KUKA KRL program: EPS_2_25694_GD02_A_20260114065900.src

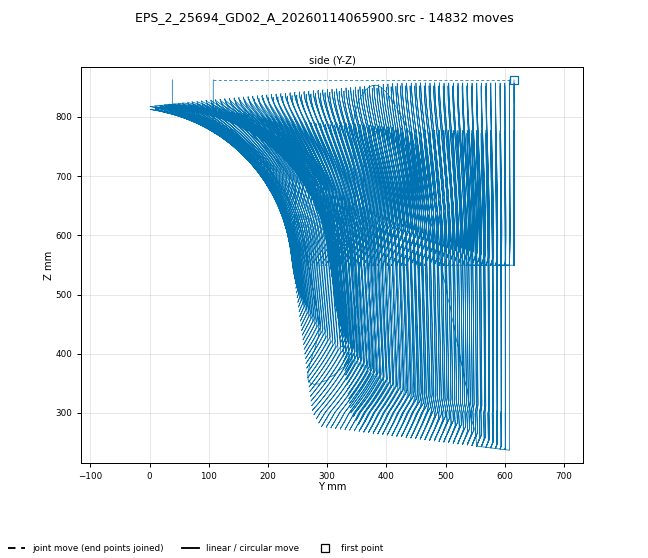
[picture p0: tool path of EPS_2_25694_GD02_A_20260114065900.src, 14832 of 14834 moves have a stored position in this frame; points joined in program order, loops and branches not executed]
&ACCESS RVP
&REL 4
&COMMENT QRS 19112012
&PARAM EDITMASK = *
DEF PART()
EXT BAS (BAS_COMMAND :IN,REAL :IN )
INT I
BAS (#INITMOV,0 )

;KUKA QRS Post kuka4.cps  Date:22-06-2017 !

File_ID=2962

QRS_PRE_INIT()

;Init var - Until changes are made in qrs_pre_init
Outlet_Square_prg=0
Inlet_1_Square_prg=0
Inlet_2_Square_prg=0
Inlet_3_Square_prg=0
Inlet_4_Square_prg=0
Inlet_5_Square_prg=0

Outlet_1={X 0.000, Y 425.000, Z 586.000, B 0.000, E1 0.000 }
Inlet_1={X 0.000, Y 466.000, Z 544.000, B 0.000, E1 154.000 }
Outlet_1_type=533
Inlet_1_type=457
;QRS#1=Sidecore dimensions
;QRS#2=525-21" Concrete
;QRS#3=450-18" Concrete
;QRS#4=
;QRS#5=
;QRS#6=
;QRS#7=
;QRS#8=
;QRS#9=S306-32
;QRS#10=28A PSX-2
;QRS#11=
;QRS#12=
;QRS#13=
;QRS#14=
;QRS#15=
;QRS#16=1220x127x1219 4'
;QRS#17=EPS Height
;QRS#18=852,5
;QRS#19=*
;QRS#20= UPDATED VERSION 22-06-2017
;QRS#21=*
Outlet_Square=0250
Inlet_1_Square=0250
Inlet_2_Square=0
Inlet_3_Square=0
Inlet_4_Square=0
Inlet_5_Square=0
Mill_Square=1
Outlet_Square_Prg=263
Inlet_1_Square_prg=274

QRS_INIT()

$ADVANCE=5

; T1
PTP {E1 172.625,E2 172.625}
PTP {X 0,Y 615.419,A -85,B 0,C 180,E1 172.625,E2 172.625,E3 0,E4 0,E5 0,E6 0}
QRS_SPEED_INIT()
LIN {X 0,Y 615.419,Z 862.5,A -85,B 0,C 180,E1 172.625,E2 172.625,E3 0,E4 0,E5 0,E6 0} C_VEL
LIN {X 0,Y 615.419,Z 551.53,A -85,B 0,C 180,E1 172.625,E2 172.625} C_VEL
LIN {X 0,Y 615.447,Z 549.53,A -85,B 0,C 180,E1 172.811,E2 172.811} C_VEL
LIN {X 0,Y 615.861,Z 549.53,A -85,B 0,C 180,E1 174.195,E2 174.195} C_VEL
LIN {X 0,Y 615.858,Z 549.53,A -85,B 0,C 180,E1 178.842,E2 178.842} C_VEL
LIN {X 0,Y 615.837,Z 549.53,A -85,B 0,C 180,E1 183.481,E2 183.481} C_VEL
LIN {X 0,Y 615.852,Z 549.53,A -85,B 0,C 180,E1 188.144,E2 188.144} C_VEL
LIN {X 0,Y 615.818,Z 549.53,A -85,B 0,C 180,E1 192.862,E2 192.862} C_VEL
LIN {X 0,Y 615.818,Z 549.53,A -85,B 0,C 180,E1 197.671,E2 197.671} C_VEL
LIN {X 0,Y 615.804,Z 549.53,A -85,B 0,C 180,E1 197.994,E2 197.994} C_VEL
LIN {X 0,Y 615.767,Z 549.53,A -85,B 0,C 180,E1 202.614,E2 202.614} C_VEL
LIN {X 0,Y 615.241,Z 549.53,A -85,B 0,C 180,E1 205.173,E2 205.173} C_VEL
LIN {X 0,Y 615.742,Z 549.53,A -85,B 0,C 180,E1 207.742,E2 207.742} C_VEL
LIN {X 0,Y 615.253,Z 549.53,A -85,B 0,C 180,E1 210.422,E2 210.422} C_VEL
LIN {X 0,Y 615.857,Z 549.53,A -85,B 0,C 180,E1 213.116,E2 213.116} C_VEL
LIN {X 0,Y 615.548,Z 549.53,A -85,B 0,C 180,E1 215.951,E2 215.951} C_VEL
LIN {X 0,Y 615.599,Z 549.53,A -85,B 0,C 180,E1 217.864,E2 217.864} C_VEL
LIN {X 0,Y 615.649,Z 549.53,A -85,B 0,C 180,E1 221.91,E2 221.91} C_VEL
LIN {X 0,Y 615.215,Z 549.53,A -85,B 0,C 180,E1 225.149,E2 225.149} C_VEL
LIN {X 0,Y 615.671,Z 549.53,A -85,B 0,C 180,E1 228.092,E2 228.092} C_VEL
LIN {X 0,Y 615.575,Z 549.53,A -85,B 0,C 180,E1 232.139,E2 232.139} C_VEL
LIN {X 0,Y 615.56,Z 549.53,A -85,B 0,C 180,E1 234.05,E2 234.05} C_VEL
LIN {X 0,Y 615.724,Z 549.53,A -85,B 0,C 180,E1 236.077,E2 236.077} C_VEL
LIN {X 0,Y 615.758,Z 549.53,A -85,B 0,C 180,E1 236.878,E2 236.878} C_VEL
LIN {X 0,Y 615.847,Z 549.53,A -85,B 0,C 180,E1 240.622,E2 240.622} C_VEL
LIN {X 0,Y 615.221,Z 549.53,A -85,B 0,C 180,E1 240.78,E2 240.78} C_VEL
LIN {X 0,Y 615.113,Z 550.032,A -85,B 0,C 180,E1 240.802,E2 240.802} C_VEL
LIN {X 0,Y 615.441,Z 600.013,A -85,B 0,C 180,E1 241.477,E2 241.477} C_VEL
LIN {X 0,Y 615.52,Z 611.103,A -85,B 0,C 180,E1 241.656,E2 241.656} C_VEL
LIN {X 0,Y 615.538,Z 625.601,A -85,B 0,C 180,E1 241.961,E2 241.961} C_VEL
LIN {X 0,Y 615.511,Z 635.884,A -85,B 0,C 180,E1 242.221,E2 242.221} C_VEL
LIN {X 0,Y 615.677,Z 651.48,A -85,B 0,C 180,E1 242.705,E2 242.705} C_VEL
LIN {X 0,Y 615.654,Z 663.918,A -85,B 0,C 180,E1 243.151,E2 243.151} C_VEL
LIN {X 0,Y 615.577,Z 673.836,A -85,B 0,C 180,E1 243.553,E2 243.553} C_VEL
LIN {X 0,Y 615.711,Z 689.57,A -85,B 0,C 180,E1 244.286,E2 244.286} C_VEL
LIN {X 0,Y 615.693,Z 701.923,A -85,B 0,C 180,E1 244.935,E2 244.935} C_VEL
LIN {X 0,Y 615.683,Z 713.602,A -85,B 0,C 180,E1 245.616,E2 245.616} C_VEL
LIN {X 0,Y 615.707,Z 725.064,A -85,B 0,C 180,E1 246.355,E2 246.355} C_VEL
LIN {X 0,Y 615.721,Z 736.37,A -85,B 0,C 180,E1 247.156,E2 247.156} C_VEL
LIN {X 0,Y 615.717,Z 747.376,A -85,B 0,C 180,E1 248.011,E2 248.011} C_VEL
LIN {X 0,Y 615.704,Z 756.639,A -85,B 0,C 180,E1 248.79,E2 248.79} C_VEL
LIN {X 0,Y 615.752,Z 766.777,A -85,B 0,C 180,E1 249.722,E2 249.722} C_VEL
LIN {X 0,Y 615.723,Z 776.042,A -85,B 0,C 180,E1 250.645,E2 250.645} C_VEL
LIN {X 0,Y 615.683,Z 784.412,A -85,B 0,C 180,E1 251.548,E2 251.548} C_VEL
LIN {X 0,Y 615.767,Z 792.766,A -85,B 0,C 180,E1 252.531,E2 252.531} C_VEL
LIN {X 0,Y 615.719,Z 800.672,A -85,B 0,C 180,E1 253.541,E2 253.541} C_VEL
LIN {X 0,Y 615.582,Z 807.418,A -85,B 0,C 180,E1 254.471,E2 254.471} C_VEL
LIN {X 0,Y 615.671,Z 815.053,A -85,B 0,C 180,E1 255.643,E2 255.643} C_VEL
LIN {X 0,Y 615.808,Z 820.43,A -85,B 0,C 180,E1 256.542,E2 256.542} C_VEL
LIN {X 0,Y 615.575,Z 826.903,A -85,B 0,C 180,E1 257.727,E2 257.727} C_VEL
LIN {X 0,Y 615.615,Z 832.619,A -85,B 0,C 180,E1 258.912,E2 258.912} C_VEL
LIN {X 0,Y 615.829,Z 837.629,A -85,B 0,C 180,E1 260.095,E2 260.095} C_VEL
LIN {X 0,Y 615.604,Z 842.059,A -85,B 0,C 180,E1 261.267,E2 261.267} C_VEL
LIN {X 0,Y 615.655,Z 846.467,A -85,B 0,C 180,E1 262.659,E2 262.659} C_VEL
LIN {X 0,Y 615.789,Z 849.367,A -85,B 0,C 180,E1 263.748,E2 263.748} C_VEL
LIN {X 0,Y 615.594,Z 851.398,A -85,B 0,C 180,E1 264.656,E2 264.656} C_VEL
LIN {X 0,Y 615.536,Z 853.159,A -85,B 0,C 180,E1 265.587,E2 265.587} C_VEL
LIN {X 0,Y 615.642,Z 854.59,A -85,B 0,C 180,E1 266.518,E2 266.518} C_VEL
LIN {X 0,Y 615.713,Z 856.053,A -85,B 0,C 180,E1 267.911,E2 267.911} C_VEL
LIN {X 0,Y 615.553,Z 856.714,A -85,B 0,C 180,E1 268.839,E2 268.839} C_VEL
LIN {X 0,Y 615.842,Z 856.659,A -85,B 0,C 180,E1 271.158,E2 271.158} C_VEL
LIN {X 0,Y 615.567,Z 855.719,A -85,B 0,C 180,E1 272.551,E2 272.551} C_VEL
LIN {X 0,Y 615.55,Z 854.61,A -85,B 0,C 180,E1 273.481,E2 273.481} C_VEL
LIN {X 0,Y 615.713,Z 853.131,A -85,B 0,C 180,E1 274.41,E2 274.41} C_VEL
LIN {X 0,Y 615.771,Z 851.372,A -85,B 0,C 180,E1 275.34,E2 275.34} C_VEL
LIN {X 0,Y 615.615,Z 849.407,A -85,B 0,C 180,E1 276.25,E2 276.25} C_VEL
LIN {X 0,Y 615.622,Z 846.269,A -85,B 0,C 180,E1 277.417,E2 277.417} C_VEL
LIN {X 0,Y 615.784,Z 842.039,A -85,B 0,C 180,E1 278.729,E2 278.729} C_VEL
LIN {X 0,Y 615.572,Z 837.675,A -85,B 0,C 180,E1 279.907,E2 279.907} C_VEL
LIN {X 0,Y 615.632,Z 832.626,A -85,B 0,C 180,E1 281.085,E2 281.085} C_VEL
LIN {X 0,Y 615.805,Z 826.888,A -85,B 0,C 180,E1 282.266,E2 282.266} C_VEL
LIN {X 0,Y 615.626,Z 820.461,A -85,B 0,C 180,E1 283.459,E2 283.459} C_VEL
LIN {X 0,Y 615.698,Z 813.201,A -85,B 0,C 180,E1 284.653,E2 284.653} C_VEL
LIN {X 0,Y 615.811,Z 807.636,A -85,B 0,C 180,E1 285.488,E2 285.488} C_VEL
LIN {X 0,Y 615.663,Z 798.205,A -85,B 0,C 180,E1 286.79,E2 286.79} C_VEL
LIN {X 0,Y 615.737,Z 789.613,A -85,B 0,C 180,E1 287.852,E2 287.852} C_VEL
LIN {X 0,Y 615.77,Z 781.421,A -85,B 0,C 180,E1 288.783,E2 288.783} C_VEL
LIN {X 0,Y 615.696,Z 771.534,A -85,B 0,C 180,E1 289.815,E2 289.815} C_VEL
LIN {X 0,Y 615.715,Z 763.548,A -85,B 0,C 180,E1 290.587,E2 290.587} C_VEL
LIN {X 0,Y 615.746,Z 753.046,A -85,B 0,C 180,E1 291.517,E2 291.517} C_VEL
LIN {X 0,Y 615.704,Z 743.056,A -85,B 0,C 180,E1 292.335,E2 292.335} C_VEL
LIN {X 0,Y 615.702,Z 733.306,A -85,B 0,C 180,E1 293.07,E2 293.07} C_VEL
LIN {X 0,Y 615.683,Z 721.643,A -85,B 0,C 180,E1 293.873,E2 293.873} C_VEL
LIN {X 0,Y 615.698,Z 709.605,A -85,B 0,C 180,E1 294.622,E2 294.622} C_VEL
LIN {X 0,Y 615.65,Z 698.907,A -85,B 0,C 180,E1 295.233,E2 295.233} C_VEL
LIN {X 0,Y 615.644,Z 688.043,A -85,B 0,C 180,E1 295.795,E2 295.795} C_VEL
LIN {X 0,Y 615.702,Z 673.896,A -85,B 0,C 180,E1 296.439,E2 296.439} C_VEL
LIN {X 0,Y 615.617,Z 660.697,A -85,B 0,C 180,E1 296.97,E2 296.97} C_VEL
LIN {X 0,Y 615.556,Z 651.549,A -85,B 0,C 180,E1 297.299,E2 297.299} C_VEL
LIN {X 0,Y 615.623,Z 634.845,A -85,B 0,C 180,E1 297.8,E2 297.8} C_VEL
LIN {X 0,Y 615.442,Z 622.425,A -85,B 0,C 180,E1 298.118,E2 298.118} C_VEL
LIN {X 0,Y 615.615,Z 610.181,A -85,B 0,C 180,E1 298.357,E2 298.357} C_VEL
LIN {X 0,Y 615.523,Z 589,A -85,B 0,C 180,E1 298.668,E2 298.668} C_VEL
LIN {X 0,Y 615.166,Z 549.53,A -85,B 0,C 180,E1 299.213,E2 299.213} C_VEL
LIN {X 0,Y 615.783,Z 549.53,A -85,B 0,C 180,E1 299.346,E2 299.346} C_VEL
LIN {X 0,Y 615.859,Z 549.53,A -85,B 0,C 180,E1 300.386,E2 300.386} C_VEL
LIN {X 0,Y 615.153,Z 549.53,A -85,B 0,C 180,E1 303.844,E2 303.844} C_VEL
LIN {X 0,Y 615.7,Z 549.53,A -85,B 0,C 180,E1 305.938,E2 305.938} C_VEL
LIN {X 0,Y 615.751,Z 549.53,A -85,B 0,C 180,E1 308.854,E2 308.854} C_VEL
LIN {X 0,Y 615.252,Z 549.53,A -85,B 0,C 180,E1 311.94,E2 311.94} C_VEL
LIN {X 0,Y 615.68,Z 549.53,A -85,B 0,C 180,E1 314.894,E2 314.894} C_VEL
LIN {X 0,Y 615.644,Z 549.53,A -85,B 0,C 180,E1 318.494,E2 318.494} C_VEL
LIN {X 0,Y 615.361,Z 549.53,A -85,B 0,C 180,E1 321.114,E2 321.114} C_VEL
LIN {X 0,Y 615.413,Z 549.53,A -85,B 0,C 180,E1 322.155,E2 322.155} C_VEL
LIN {X 0,Y 615.665,Z 549.53,A -85,B 0,C 180,E1 324.057,E2 324.057} C_VEL
LIN {X 0,Y 615.125,Z 549.53,A -85,B 0,C 180,E1 326.84,E2 326.84} C_VEL
LIN {X 0,Y 615.717,Z 549.53,A -85,B 0,C 180,E1 329.603,E2 329.603} C_VEL
LIN {X 0,Y 615.208,Z 549.53,A -85,B 0,C 180,E1 332.232,E2 332.232} C_VEL
LIN {X 0,Y 615.747,Z 549.53,A -85,B 0,C 180,E1 334.849,E2 334.849} C_VEL
LIN {X 0,Y 615.78,Z 549.53,A -85,B 0,C 180,E1 339.877,E2 339.877} C_VEL
LIN {X 0,Y 615.794,Z 549.53,A -85,B 0,C 180,E1 343.783,E2 343.783} C_VEL
LIN {X 0,Y 615.811,Z 549.53,A -85,B 0,C 180,E1 349.506,E2 349.506} C_VEL
LIN {X 0,Y 615.84,Z 549.53,A -85,B 0,C 180,E1 354.192,E2 354.192} C_VEL
LIN {X 0,Y 615.881,Z 549.53,A -85,B 0,C 180,E1 358.839,E2 358.839} C_VEL
LIN {X 0,Y 615.868,Z 549.53,A -85,B 0,C 180,E1 363.479,E2 363.479} C_VEL
LIN {X 0,Y 615.819,Z 549.53,A -85,B 0,C 180,E1 368.142,E2 368.142} C_VEL
LIN {X 0,Y 615.829,Z 549.53,A -85,B 0,C 180,E1 372.86,E2 372.86} C_VEL
LIN {X 0,Y 615.811,Z 549.53,A -85,B 0,C 180,E1 377.669,E2 377.669} C_VEL
LIN {X 0,Y 615.807,Z 549.53,A -85,B 0,C 180,E1 378.001,E2 378.001} C_VEL
LIN {X 0,Y 615.775,Z 549.53,A -85,B 0,C 180,E1 382.611,E2 382.611} C_VEL
LIN {X 0,Y 615.234,Z 549.53,A -85,B 0,C 180,E1 385.171,E2 385.171} C_VEL
LIN {X 0,Y 615.726,Z 549.53,A -85,B 0,C 180,E1 387.74,E2 387.74} C_VEL
LIN {X 0,Y 615.245,Z 549.53,A -85,B 0,C 180,E1 390.42,E2 390.42} C_VEL
LIN {X 0,Y 615.861,Z 549.53,A -85,B 0,C 180,E1 393.113,E2 393.113} C_VEL
LIN {X 0,Y 615.544,Z 549.53,A -85,B 0,C 180,E1 395.949,E2 395.949} C_VEL
LIN {X 0,Y 615.616,Z 549.53,A -85,B 0,C 180,E1 397.87,E2 397.87} C_VEL
LIN {X 0,Y 615.686,Z 549.53,A -85,B 0,C 180,E1 401.904,E2 401.904} C_VEL
LIN {X 0,Y 615.226,Z 549.53,A -85,B 0,C 180,E1 405.145,E2 405.145} C_VEL
LIN {X 0,Y 615.687,Z 549.53,A -85,B 0,C 180,E1 408.096,E2 408.096} C_VEL
LIN {X 0,Y 615.59,Z 549.53,A -85,B 0,C 180,E1 412.133,E2 412.133} C_VEL
LIN {X 0,Y 615.555,Z 549.53,A -85,B 0,C 180,E1 414.052,E2 414.052} C_VEL
LIN {X 0,Y 615.724,Z 549.53,A -85,B 0,C 180,E1 416.073,E2 416.073} C_VEL
LIN {X 0,Y 615.732,Z 549.53,A -85,B 0,C 180,E1 416.879,E2 416.879} C_VEL
LIN {X 0,Y 615.544,Z 549.53,A -85,B 0,C 180,E1 420.514,E2 420.514} C_VEL
LIN {X 0,Y 615.505,Z 549.53,A -85,B 0,C 180,E1 422.249,E2 422.249} C_VEL
LIN {X 0,Y 615.421,Z 549.53,A -85,B 0,C 180,E1 425.664,E2 425.664} C_VEL
LIN {X 0,Y 615.586,Z 549.53,A -85,B 0,C 180,E1 427.382,E2 427.382} C_VEL
LIN {X 0,Y 615.803,Z 549.53,A -85,B 0,C 180,E1 431.999,E2 431.999} C_VEL
LIN {X 0,Y 615.813,Z 549.53,A -85,B 0,C 180,E1 432.331,E2 432.331} C_VEL
LIN {X 0,Y 615.817,Z 549.53,A -85,B 0,C 180,E1 437.14,E2 437.14} C_VEL
LIN {X 0,Y 615.839,Z 549.53,A -85,B 0,C 180,E1 441.858,E2 441.858} C_VEL
LIN {X 0,Y 615.871,Z 549.53,A -85,B 0,C 180,E1 446.521,E2 446.521} C_VEL
LIN {X 0,Y 615.493,Z 549.53,A -85,B 0,C 180,E1 448.841,E2 448.841} C_VEL
LIN {X 0,Y 615.592,Z 549.53,A -85,B 0,C 180,E1 451.161,E2 451.161} C_VEL
LIN {X 0,Y 615.322,Z 549.53,A -85,B 0,C 180,E1 451.292,E2 451.292} C_VEL
LIN {X 0,Y 615.521,Z 551.584,A -85,B 0,C 180,E1 451.335,E2 451.335} C_VEL
LIN {X 0,Y 615.568,Z 564.334,A -85,B 0,C 180,E1 451.538,E2 451.538} C_VEL
LIN {X 0,Y 615.674,Z 576.042,A -85,B 0,C 180,E1 451.784,E2 451.784} C_VEL
LIN {X 0,Y 615.724,Z 587.841,A -85,B 0,C 180,E1 452.089,E2 452.089} C_VEL
LIN {X 0,Y 615.604,Z 599.369,A -85,B 0,C 180,E1 452.437,E2 452.437} C_VEL
LIN {X 0,Y 615.735,Z 610.571,A -85,B 0,C 180,E1 452.843,E2 452.843} C_VEL
LIN {X 0,Y 615.763,Z 621.858,A -85,B 0,C 180,E1 453.307,E2 453.307} C_VEL
LIN {X 0,Y 615.701,Z 631.978,A -85,B 0,C 180,E1 453.773,E2 453.773} C_VEL
LIN {X 0,Y 615.733,Z 642.117,A -85,B 0,C 180,E1 454.295,E2 454.295} C_VEL
LIN {X 0,Y 615.752,Z 652.294,A -85,B 0,C 180,E1 454.877,E2 454.877} C_VEL
LIN {X 0,Y 615.751,Z 663.293,A -85,B 0,C 180,E1 455.576,E2 455.576} C_VEL
LIN {X 0,Y 615.738,Z 671.827,A -85,B 0,C 180,E1 456.167,E2 456.167} C_VEL
LIN {X 0,Y 615.744,Z 681.127,A -85,B 0,C 180,E1 456.874,E2 456.874} C_VEL
LIN {X 0,Y 615.757,Z 689.335,A -85,B 0,C 180,E1 457.55,E2 457.55} C_VEL
LIN {X 0,Y 615.801,Z 697.599,A -85,B 0,C 180,E1 458.291,E2 458.291} C_VEL
LIN {X 0,Y 615.737,Z 706.589,A -85,B 0,C 180,E1 459.172,E2 459.172} C_VEL
LIN {X 0,Y 615.734,Z 713.495,A -85,B 0,C 180,E1 459.907,E2 459.907} C_VEL
LIN {X 0,Y 615.829,Z 721.068,A -85,B 0,C 180,E1 460.789,E2 460.789} C_VEL
LIN {X 0,Y 615.72,Z 728.094,A -85,B 0,C 180,E1 461.677,E2 461.677} C_VEL
LIN {X 0,Y 615.671,Z 734.517,A -85,B 0,C 180,E1 462.568,E2 462.568} C_VEL
LIN {X 0,Y 615.768,Z 740.348,A -85,B 0,C 180,E1 463.459,E2 463.459} C_VEL
LIN {X 0,Y 615.748,Z 745.727,A -85,B 0,C 180,E1 464.355,E2 464.355} C_VEL
LIN {X 0,Y 615.626,Z 750.659,A -85,B 0,C 180,E1 465.258,E2 465.258} C_VEL
LIN {X 0,Y 615.725,Z 756.396,A -85,B 0,C 180,E1 466.459,E2 466.459} C_VEL
LIN {X 0,Y 615.801,Z 759.837,A -85,B 0,C 180,E1 467.266,E2 467.266} C_VEL
LIN {X 0,Y 615.629,Z 764.32,A -85,B 0,C 180,E1 468.452,E2 468.452} C_VEL
LIN {X 0,Y 615.688,Z 767.676,A -85,B 0,C 180,E1 469.51,E2 469.51} C_VEL
LIN {X 0,Y 615.806,Z 769.293,A -85,B 0,C 180,E1 470.122,E2 470.122} C_VEL
LIN {X 0,Y 615.749,Z 770.875,A -85,B 0,C 180,E1 470.743,E2 470.743} C_VEL
LIN {X 0,Y 615.585,Z 773.45,A -85,B 0,C 180,E1 471.994,E2 471.994} C_VEL
LIN {X 0,Y 615.622,Z 774.496,A -85,B 0,C 180,E1 472.619,E2 472.619} C_VEL
LIN {X 0,Y 615.769,Z 775.581,A -85,B 0,C 180,E1 473.516,E2 473.516} C_VEL
LIN {X 0,Y 615.695,Z 776.356,A -85,B 0,C 180,E1 474.392,E2 474.392} C_VEL
LIN {X 0,Y 615.585,Z 776.792,A -85,B 0,C 180,E1 475.158,E2 475.158} C_VEL
LIN {X 0,Y 615.649,Z 776.852,A -85,B 0,C 180,E1 476.443,E2 476.443} C_VEL
LIN {X 0,Y 615.764,Z 776.185,A -85,B 0,C 180,E1 477.74,E2 477.74} C_VEL
LIN {X 0,Y 615.646,Z 775.322,A -85,B 0,C 180,E1 478.631,E2 478.631} C_VEL
LIN {X 0,Y 615.648,Z 774.08,A -85,B 0,C 180,E1 479.534,E2 479.534} C_VEL
LIN {X 0,Y 615.799,Z 772.553,A -85,B 0,C 180,E1 480.392,E2 480.392} C_VEL
LIN {X 0,Y 615.717,Z 770.538,A -85,B 0,C 180,E1 481.325,E2 481.325} C_VEL
LIN {X 0,Y 615.599,Z 768.043,A -85,B 0,C 180,E1 482.27,E2 482.27} C_VEL
LIN {X 0,Y 615.707,Z 763.994,A -85,B 0,C 180,E1 483.548,E2 483.548} C_VEL
LIN {X 0,Y 615.783,Z 760.587,A -85,B 0,C 180,E1 484.456,E2 484.456} C_VEL
LIN {X 0,Y 615.616,Z 755.31,A -85,B 0,C 180,E1 485.698,E2 485.698} C_VEL
LIN {X 0,Y 615.727,Z 749.175,A -85,B 0,C 180,E1 486.921,E2 486.921} C_VEL
LIN {X 0,Y 615.826,Z 745.732,A -85,B 0,C 180,E1 487.551,E2 487.551} C_VEL
LIN {X 0,Y 615.668,Z 739.293,A -85,B 0,C 180,E1 488.626,E2 488.626} C_VEL
LIN {X 0,Y 615.685,Z 733.233,A -85,B 0,C 180,E1 489.533,E2 489.533} C_VEL
LIN {X 0,Y 615.809,Z 725.413,A -85,B 0,C 180,E1 490.581,E2 490.581} C_VEL
LIN {X 0,Y 615.706,Z 717.809,A -85,B 0,C 180,E1 491.512,E2 491.512} C_VEL
LIN {X 0,Y 615.692,Z 710.996,A -85,B 0,C 180,E1 492.278,E2 492.278} C_VEL
LIN {X 0,Y 615.759,Z 703.806,A -85,B 0,C 180,E1 493.022,E2 493.022} C_VEL
LIN {X 0,Y 615.754,Z 694.645,A -85,B 0,C 180,E1 493.889,E2 493.889} C_VEL
LIN {X 0,Y 615.725,Z 686.193,A -85,B 0,C 180,E1 494.624,E2 494.624} C_VEL
LIN {X 0,Y 615.738,Z 677.048,A -85,B 0,C 180,E1 495.352,E2 495.352} C_VEL
LIN {X 0,Y 615.745,Z 668.071,A -85,B 0,C 180,E1 496.009,E2 496.009} C_VEL
LIN {X 0,Y 615.751,Z 658.065,A -85,B 0,C 180,E1 496.675,E2 496.675} C_VEL
LIN {X 0,Y 615.747,Z 648.614,A -85,B 0,C 180,E1 497.249,E2 497.249} C_VEL
LIN {X 0,Y 615.67,Z 638.444,A -85,B 0,C 180,E1 497.812,E2 497.812} C_VEL
LIN {X 0,Y 615.756,Z 627.627,A -85,B 0,C 180,E1 498.343,E2 498.343} C_VEL
LIN {X 0,Y 615.751,Z 616.912,A -85,B 0,C 180,E1 498.815,E2 498.815} C_VEL
LIN {X 0,Y 615.675,Z 606.253,A -85,B 0,C 180,E1 499.232,E2 499.232} C_VEL
LIN {X 0,Y 615.684,Z 596.594,A -85,B 0,C 180,E1 499.564,E2 499.564} C_VEL
LIN {X 0,Y 615.68,Z 583.685,A -85,B 0,C 180,E1 499.938,E2 499.938} C_VEL
LIN {X 0,Y 615.56,Z 573.065,A -85,B 0,C 180,E1 500.2,E2 500.2} C_VEL
LIN {X 0,Y 615.621,Z 560.618,A -85,B 0,C 180,E1 500.436,E2 500.436} C_VEL
LIN {X 0,Y 615.473,Z 550.692,A -85,B 0,C 180,E1 500.59,E2 500.59} C_VEL
LIN {X 0,Y 615.123,Z 549.53,A -85,B 0,C 180,E1 500.623,E2 500.623} C_VEL
LIN {X 0,Y 615.755,Z 549.53,A -85,B 0,C 180,E1 500.83,E2 500.83} C_VEL
LIN {X 0,Y 615.851,Z 549.53,A -85,B 0,C 180,E1 501.154,E2 501.154} C_VEL
LIN {X 0,Y 615.701,Z 549.53,A -85,B 0,C 180,E1 504.062,E2 504.062} C_VEL
LIN {X 0,Y 615.123,Z 549.53,A -85,B 0,C 180,E1 506.842,E2 506.842} C_VEL
LIN {X 0,Y 615.677,Z 549.53,A -85,B 0,C 180,E1 509.604,E2 509.604} C_VEL
LIN {X 0,Y 615.181,Z 549.53,A -85,B 0,C 180,E1 512.234,E2 512.234} C_VEL
LIN {X 0,Y 615.722,Z 549.53,A -85,B 0,C 180,E1 514.85,E2 514.85} C_VEL
LIN {X 0,Y 615.796,Z 549.53,A -85,B 0,C 180,E1 519.88,E2 519.88} C_VEL
LIN {X 0,Y 615.742,Z 549.53,A -85,B 0,C 180,E1 523.3,E2 523.3} C_VEL
LIN {X 0,Y 615.403,Z 549.53,A -85,B 0,C 180,E1 524.739,E2 524.739} C_VEL
LIN {X 0,Y 615.803,Z 549.53,A -85,B 0,C 180,E1 529.508,E2 529.508} C_VEL
LIN {X 0,Y 615.447,Z 549.53,A -85,B 0,C 180,E1 532.811,E2 532.811} C_VEL
LIN {X 0,Y 613.027,Z 549.53,A -85,B 0,C 180,E1 534.013,E2 534.013} C_VEL
LIN {X 0,Y 607.603,Z 549.53,A -85,B 0,C 180,E1 535.81,E2 535.81} C_VEL
LIN {X 0,Y 607.492,Z 549.53,A -85,B 0,C 180,E1 536.018,E2 536.018} C_VEL
LIN {X 0,Y 607.6,Z 549.53,A -85,B 0,C 180,E1 540.012,E2 540.012} C_VEL
LIN {X 0,Y 607.677,Z 549.53,A -85,B 0,C 180,E1 544.283,E2 544.283} C_VEL
LIN {X 0,Y 607.793,Z 549.53,A -85,B 0,C 180,E1 548.577,E2 548.577} C_VEL
LIN {X 0,Y 607.905,Z 549.53,A -85,B 0,C 180,E1 552.918,E2 552.918} C_VEL
LIN {X 0,Y 607.624,Z 549.53,A -85,B 0,C 180,E1 558.843,E2 558.843} C_VEL
LIN {X 0,Y 607.589,Z 549.53,A -85,B 0,C 180,E1 563.421,E2 563.421} C_VEL
LIN {X 0,Y 607.697,Z 549.53,A -85,B 0,C 180,E1 568.157,E2 568.157} C_VEL
LIN {X 0,Y 607.956,Z 549.53,A -85,B 0,C 180,E1 573.103,E2 573.103} C_VEL
LIN {X 0,Y 607.549,Z 549.53,A -85,B 0,C 180,E1 578.389,E2 578.389} C_VEL
LIN {X 0,Y 607.671,Z 549.53,A -85,B 0,C 180,E1 582.108,E2 582.108} C_VEL
LIN {X 0,Y 607.743,Z 549.53,A -85,B 0,C 180,E1 588.153,E2 588.153} C_VEL
LIN {X 0,Y 607.597,Z 549.53,A -85,B 0,C 180,E1 593.413,E2 593.413} C_VEL
LIN {X 0,Y 607.685,Z 549.53,A -85,B 0,C 180,E1 597.597,E2 597.597} C_VEL
LIN {X 0,Y 607.878,Z 549.53,A -85,B 0,C 180,E1 600.413,E2 600.413} C_VEL
LIN {X 0,Y 608.594,Z 622.659,A -85,B 0,C 180,E1 601.542,E2 601.542} C_VEL
LIN {X 0,Y 608.564,Z 661.909,A -85,B 0,C 180,E1 602.735,E2 602.735} C_VEL
LIN {X 0,Y 608.417,Z 699.451,A -85,B 0,C 180,E1 604.474,E2 604.474} C_VEL
LIN {X 0,Y 608.262,Z 735.694,A -85,B 0,C 180,E1 606.808,E2 606.808} C_VEL
LIN {X 0,Y 608.119,Z 767.053,A -85,B 0,C 180,E1 609.483,E2 609.483} C_VEL
LIN {X 0,Y 608.025,Z 794.243,A -85,B 0,C 180,E1 612.488,E2 612.488} C_VEL
LIN {X 0,Y 607.886,Z 817.261,A -85,B 0,C 180,E1 615.811,E2 615.811} C_VEL
LIN {X 0,Y 607.819,Z 834.982,A -85,B 0,C 180,E1 619.27,E2 619.27} C_VEL
LIN {X 0,Y 607.792,Z 847.68,A -85,B 0,C 180,E1 622.87,E2 622.87} C_VEL
LIN {X 0,Y 607.673,Z 853.958,A -85,B 0,C 180,E1 625.729,E2 625.729} C_VEL
LIN {X 0,Y 607.712,Z 857.086,A -85,B 0,C 180,E1 628.578,E2 628.578} C_VEL
LIN {X 0,Y 607.885,Z 857.085,A -85,B 0,C 180,E1 631.424,E2 631.424} C_VEL
LIN {X 0,Y 607.861,Z 852.755,A -85,B 0,C 180,E1 634.986,E2 634.986} C_VEL
LIN {X 0,Y 607.879,Z 842.068,A -85,B 0,C 180,E1 638.927,E2 638.927} C_VEL
LIN {X 0,Y 607.905,Z 826.444,A -85,B 0,C 180,E1 642.546,E2 642.546} C_VEL
LIN {X 0,Y 607.958,Z 805.34,A -85,B 0,C 180,E1 646.031,E2 646.031} C_VEL
LIN {X 0,Y 608.034,Z 779.208,A -85,B 0,C 180,E1 649.269,E2 649.269} C_VEL
LIN {X 0,Y 608.172,Z 749.008,A -85,B 0,C 180,E1 652.139,E2 652.139} C_VEL
LIN {X 0,Y 608.319,Z 715.869,A -85,B 0,C 180,E1 654.552,E2 654.552} C_VEL
LIN {X 0,Y 608.482,Z 679.714,A -85,B 0,C 180,E1 656.514,E2 656.514} C_VEL
LIN {X 0,Y 608.576,Z 642.95,A -85,B 0,C 180,E1 657.911,E2 657.911} C_VEL
LIN {X 0,Y 608.666,Z 607.028,A -85,B 0,C 180,E1 658.76,E2 658.76} C_VEL
LIN {X 0,Y 607.895,Z 549.53,A -85,B 0,C 180,E1 659.62,E2 659.62} C_VEL
LIN {X 0,Y 607.678,Z 549.53,A -85,B 0,C 180,E1 666.584,E2 666.584} C_VEL
LIN {X 0,Y 607.357,Z 549.53,A -85,B 0,C 180,E1 671.807,E2 671.807} C_VEL
LIN {X 0,Y 607.516,Z 549.53,A -85,B 0,C 180,E1 676.084,E2 676.084} C_VEL
LIN {X 0,Y 607.437,Z 549.53,A -85,B 0,C 180,E1 680.365,E2 680.365} C_VEL
LIN {X 0,Y 607.404,Z 549.53,A -85,B 0,C 180,E1 685.147,E2 685.147} C_VEL
LIN {X 0,Y 607.532,Z 549.53,A -85,B 0,C 180,E1 690.385,E2 690.385} C_VEL
LIN {X 0,Y 607.788,Z 549.53,A -85,B 0,C 180,E1 695.028,E2 695.028} C_VEL
LIN {X 0,Y 607.575,Z 549.53,A -85,B 0,C 180,E1 701.155,E2 701.155} C_VEL
LIN {X 0,Y 607.247,Z 549.53,A -85,B 0,C 180,E1 705.602,E2 705.602} C_VEL
LIN {X 0,Y 607.743,Z 549.53,A -85,B 0,C 180,E1 709.981,E2 709.981} C_VEL
LIN {X 0,Y 607.907,Z 549.53,A -85,B 0,C 180,E1 714.291,E2 714.291} C_VEL
LIN {X 0,Y 607.602,Z 549.53,A -85,B 0,C 180,E1 719.988,E2 719.988} C_VEL
LIN {X 0,Y 607.675,Z 549.53,A -85,B 0,C 180,E1 724.259,E2 724.259} C_VEL
LIN {X 0,Y 607.778,Z 549.53,A -85,B 0,C 180,E1 728.553,E2 728.553} C_VEL
LIN {X 0,Y 607.908,Z 549.53,A -85,B 0,C 180,E1 732.894,E2 732.894} C_VEL
LIN {X 0,Y 607.616,Z 549.53,A -85,B 0,C 180,E1 738.819,E2 738.819} C_VEL
LIN {X 0,Y 607.575,Z 549.53,A -85,B 0,C 180,E1 743.396,E2 743.396} C_VEL
LIN {X 0,Y 607.677,Z 549.53,A -85,B 0,C 180,E1 748.132,E2 748.132} C_VEL
LIN {X 0,Y 607.936,Z 549.53,A -85,B 0,C 180,E1 753.076,E2 753.076} C_VEL
LIN {X 0,Y 607.574,Z 549.53,A -85,B 0,C 180,E1 758.357,E2 758.357} C_VEL
LIN {X 0,Y 607.736,Z 549.53,A -85,B 0,C 180,E1 762.071,E2 762.071} C_VEL
LIN {X 0,Y 607.784,Z 549.53,A -85,B 0,C 180,E1 768.113,E2 768.113} C_VEL
LIN {X 0,Y 607.609,Z 549.53,A -85,B 0,C 180,E1 773.411,E2 773.411} C_VEL
LIN {X 0,Y 607.606,Z 549.53,A -85,B 0,C 180,E1 777.565,E2 777.565} C_VEL
LIN {X 0,Y 607.575,Z 549.53,A -85,B 0,C 180,E1 781.841,E2 781.841} C_VEL
LIN {X 0,Y 607.482,Z 549.53,A -85,B 0,C 180,E1 788.122,E2 788.122} C_VEL
LIN {X 0,Y 607.788,Z 549.53,A -85,B 0,C 180,E1 792.665,E2 792.665} C_VEL
LIN {X 0,Y 607.888,Z 549.53,A -85,B 0,C 180,E1 797.089,E2 797.089} C_VEL
LIN {X 0,Y 607.616,Z 549.53,A -85,B 0,C 180,E1 802.866,E2 802.866} C_VEL
LIN {X 0,Y 607.773,Z 549.53,A -85,B 0,C 180,E1 807.153,E2 807.153} C_VEL
LIN {X 0,Y 607.691,Z 550.216,A -85,B 0,C 180,E1 810.977,E2 810.977} C_VEL
LIN {X 0,Y 608.468,Z 588.971,A -85,B 0,C 180,E1 811.82,E2 811.82} C_VEL
LIN {X 0,Y 608.369,Z 623.891,A -85,B 0,C 180,E1 813.109,E2 813.109} C_VEL
LIN {X 0,Y 608.247,Z 656.857,A -85,B 0,C 180,E1 814.891,E2 814.891} C_VEL
LIN {X 0,Y 608.107,Z 688.902,A -85,B 0,C 180,E1 817.271,E2 817.271} C_VEL
LIN {X 0,Y 607.988,Z 716.168,A -85,B 0,C 180,E1 820.004,E2 820.004} C_VEL
LIN {X 0,Y 607.909,Z 739.215,A -85,B 0,C 180,E1 823.091,E2 823.091} C_VEL
LIN {X 0,Y 607.858,Z 756.17,A -85,B 0,C 180,E1 826.216,E2 826.216} C_VEL
LIN {X 0,Y 607.888,Z 769.2,A -85,B 0,C 180,E1 829.84,E2 829.84} C_VEL
LIN {X 0,Y 607.88,Z 776.024,A -85,B 0,C 180,E1 833.401,E2 833.401} C_VEL
LIN {X 0,Y 607.775,Z 777.334,A -85,B 0,C 180,E1 836.695,E2 836.695} C_VEL
LIN {X 0,Y 607.797,Z 774.256,A -85,B 0,C 180,E1 839.771,E2 839.771} C_VEL
LIN {X 0,Y 607.782,Z 766.115,A -85,B 0,C 180,E1 843.107,E2 843.107} C_VEL
LIN {X 0,Y 607.8,Z 753.079,A -85,B 0,C 180,E1 846.338,E2 846.338} C_VEL
LIN {X 0,Y 607.852,Z 734.699,A -85,B 0,C 180,E1 849.504,E2 849.504} C_VEL
LIN {X 0,Y 607.982,Z 710.372,A -85,B 0,C 180,E1 852.557,E2 852.557} C_VEL
LIN {X 0,Y 608.109,Z 682.965,A -85,B 0,C 180,E1 855.134,E2 855.134} C_VEL
LIN {X 0,Y 608.261,Z 650.212,A -85,B 0,C 180,E1 857.434,E2 857.434} C_VEL
LIN {X 0,Y 608.395,Z 615.362,A -85,B 0,C 180,E1 859.17,E2 859.17} C_VEL
LIN {X 0,Y 608.397,Z 579.809,A -85,B 0,C 180,E1 860.34,E2 860.34} C_VEL
LIN {X 0,Y 607.896,Z 549.53,A -85,B 0,C 180,E1 860.984,E2 860.984} C_VEL
LIN {X 0,Y 607.41,Z 549.53,A -85,B 0,C 180,E1 865.176,E2 865.176} C_VEL
LIN {X 0,Y 607.492,Z 549.53,A -85,B 0,C 180,E1 870.387,E2 870.387} C_VEL
LIN {X 0,Y 607.738,Z 549.53,A -85,B 0,C 180,E1 875.051,E2 875.051} C_VEL
LIN {X 0,Y 607.647,Z 549.53,A -85,B 0,C 180,E1 881.182,E2 881.182} C_VEL
LIN {X 0,Y 607.235,Z 549.53,A -85,B 0,C 180,E1 885.732,E2 885.732} C_VEL
LIN {X 0,Y 607.729,Z 549.53,A -85,B 0,C 180,E1 890.005,E2 890.005} C_VEL
LIN {X 0,Y 607.91,Z 549.53,A -85,B 0,C 180,E1 894.315,E2 894.315} C_VEL
LIN {X 0,Y 607.492,Z 549.53,A -85,B 0,C 180,E1 896.018,E2 896.018} C_VEL
LIN {X 0,Y 603.687,Z 549.53,A -85,B 0,C 180,E1 897.629,E2 897.629} C_VEL
LIN {X 0,Y 599.79,Z 549.53,A -85,B 0,C 180,E1 899.261,E2 899.261} C_VEL
LIN {X 0,Y 599.759,Z 549.53,A -85,B 0,C 180,E1 904.34,E2 904.34} C_VEL
LIN {X 0,Y 599.85,Z 549.53,A -85,B 0,C 180,E1 908.691,E2 908.691} C_VEL
LIN {X 0,Y 599.927,Z 549.53,A -85,B 0,C 180,E1 913.093,E2 913.093} C_VEL
LIN {X 0,Y 599.668,Z 549.53,A -85,B 0,C 180,E1 919.103,E2 919.103} C_VEL
LIN {X 0,Y 599.598,Z 549.53,A -85,B 0,C 180,E1 923.753,E2 923.753} C_VEL
LIN {X 0,Y 599.693,Z 549.53,A -85,B 0,C 180,E1 928.568,E2 928.568} C_VEL
LIN {X 0,Y 599.835,Z 549.53,A -85,B 0,C 180,E1 933.884,E2 933.884} C_VEL
LIN {X 0,Y 599.534,Z 549.53,A -85,B 0,C 180,E1 938.999,E2 938.999} C_VEL
LIN {X 0,Y 599.463,Z 549.53,A -85,B 0,C 180,E1 943.114,E2 943.114} C_VEL
LIN {X 0,Y 599.571,Z 549.53,A -85,B 0,C 180,E1 949.129,E2 949.129} C_VEL
LIN {X 0,Y 599.699,Z 549.53,A -85,B 0,C 180,E1 954.639,E2 954.639} C_VEL
LIN {X 0,Y 599.858,Z 549.678,A -85,B 0,C 180,E1 959.979,E2 959.979} C_VEL
LIN {X 0,Y 601.393,Z 557.513,A -85,B 0,C 180,E1 960.169,E2 960.169} C_VEL
LIN {X 0,Y 601.624,Z 623.673,A -85,B 0,C 180,E1 961.204,E2 961.204} C_VEL
LIN {X 0,Y 601.462,Z 662.722,A -85,B 0,C 180,E1 962.416,E2 962.416} C_VEL
LIN {X 0,Y 601.136,Z 701.22,A -85,B 0,C 180,E1 964.243,E2 964.243} C_VEL
LIN {X 0,Y 600.766,Z 736.777,A -85,B 0,C 180,E1 966.586,E2 966.586} C_VEL
LIN {X 0,Y 600.496,Z 767.704,A -85,B 0,C 180,E1 969.276,E2 969.276} C_VEL
LIN {X 0,Y 600.277,Z 795.709,A -85,B 0,C 180,E1 972.444,E2 972.444} C_VEL
LIN {X 0,Y 600.066,Z 818.366,A -85,B 0,C 180,E1 975.81,E2 975.81} C_VEL
LIN {X 0,Y 599.963,Z 835.883,A -85,B 0,C 180,E1 979.342,E2 979.342} C_VEL
LIN {X 0,Y 599.888,Z 847.68,A -85,B 0,C 180,E1 982.776,E2 982.776} C_VEL
LIN {X 0,Y 599.787,Z 853.958,A -85,B 0,C 180,E1 985.672,E2 985.672} C_VEL
LIN {X 0,Y 599.811,Z 857.087,A -85,B 0,C 180,E1 988.559,E2 988.559} C_VEL
LIN {X 0,Y 599.979,Z 857.085,A -85,B 0,C 180,E1 991.442,E2 991.442} C_VEL
LIN {X 0,Y 599.957,Z 852.755,A -85,B 0,C 180,E1 995.051,E2 995.051} C_VEL
LIN {X 0,Y 599.978,Z 842.069,A -85,B 0,C 180,E1 999.045,E2 999.045} C_VEL
LIN {X 0,Y 600.041,Z 826.445,A -85,B 0,C 180,E1 1002.713,E2 1002.713} C_VEL
LIN {X 0,Y 600.117,Z 804.714,A -85,B 0,C 180,E1 1006.334,E2 1006.334} C_VEL
LIN {X 0,Y 600.356,Z 779.069,A -85,B 0,C 180,E1 1009.541,E2 1009.541} C_VEL
LIN {X 0,Y 600.641,Z 748.452,A -85,B 0,C 180,E1 1012.479,E2 1012.479} C_VEL
LIN {X 0,Y 600.988,Z 713.92,A -85,B 0,C 180,E1 1015,E2 1015} C_VEL
LIN {X 0,Y 601.372,Z 675.861,A -85,B 0,C 180,E1 1017.035,E2 1017.035} C_VEL
LIN {X 0,Y 601.583,Z 636.494,A -85,B 0,C 180,E1 1018.465,E2 1018.465} C_VEL
LIN {X 0,Y 601.776,Z 597.397,A -85,B 0,C 180,E1 1019.274,E2 1019.274} C_VEL
LIN {X 0,Y 600.803,Z 553.114,A -85,B 0,C 180,E1 1019.922,E2 1019.922} C_VEL
LIN {X 0,Y 599.9,Z 549.53,A -85,B 0,C 180,E1 1020.023,E2 1020.023} C_VEL
LIN {X 0,Y 599.745,Z 549.53,A -85,B 0,C 180,E1 1027.148,E2 1027.148} C_VEL
LIN {X 0,Y 599.427,Z 549.53,A -85,B 0,C 180,E1 1033.106,E2 1033.106} C_VEL
LIN {X 0,Y 599.591,Z 549.53,A -85,B 0,C 180,E1 1039.029,E2 1039.029} C_VEL
LIN {X 0,Y 599.529,Z 549.53,A -85,B 0,C 180,E1 1044.621,E2 1044.621} C_VEL
LIN {X 0,Y 599.614,Z 549.53,A -85,B 0,C 180,E1 1049.774,E2 1049.774} C_VEL
LIN {X 0,Y 599.854,Z 549.53,A -85,B 0,C 180,E1 1054.911,E2 1054.911} C_VEL
LIN {X 0,Y 599.731,Z 549.53,A -85,B 0,C 180,E1 1060.899,E2 1060.899} C_VEL
LIN {X 0,Y 599.385,Z 549.53,A -85,B 0,C 180,E1 1065.409,E2 1065.409} C_VEL
LIN {X 0,Y 599.802,Z 549.53,A -85,B 0,C 180,E1 1069.847,E2 1069.847} C_VEL
LIN {X 0,Y 600.006,Z 549.53,A -85,B 0,C 180,E1 1074.216,E2 1074.216} C_VEL
LIN {X 0,Y 599.701,Z 549.53,A -85,B 0,C 180,E1 1079.988,E2 1079.988} C_VEL
LIN {X 0,Y 599.757,Z 549.53,A -85,B 0,C 180,E1 1084.316,E2 1084.316} C_VEL
LIN {X 0,Y 599.835,Z 549.53,A -85,B 0,C 180,E1 1088.667,E2 1088.667} C_VEL
LIN {X 0,Y 599.932,Z 549.53,A -85,B 0,C 180,E1 1093.068,E2 1093.068} C_VEL
LIN {X 0,Y 599.667,Z 549.53,A -85,B 0,C 180,E1 1099.078,E2 1099.078} C_VEL
LIN {X 0,Y 599.589,Z 549.53,A -85,B 0,C 180,E1 1103.727,E2 1103.727} C_VEL
LIN {X 0,Y 599.658,Z 549.53,A -85,B 0,C 180,E1 1108.542,E2 1108.542} C_VEL
LIN {X 0,Y 599.817,Z 549.53,A -85,B 0,C 180,E1 1113.878,E2 1113.878} C_VEL
LIN {X 0,Y 599.565,Z 549.53,A -85,B 0,C 180,E1 1118.966,E2 1118.966} C_VEL
LIN {X 0,Y 599.497,Z 549.53,A -85,B 0,C 180,E1 1123.115,E2 1123.115} C_VEL
LIN {X 0,Y 599.582,Z 549.53,A -85,B 0,C 180,E1 1129.127,E2 1129.127} C_VEL
LIN {X 0,Y 599.704,Z 549.53,A -85,B 0,C 180,E1 1134.637,E2 1134.637} C_VEL
LIN {X 0,Y 599.591,Z 549.53,A -85,B 0,C 180,E1 1139.777,E2 1139.777} C_VEL
LIN {X 0,Y 599.492,Z 549.53,A -85,B 0,C 180,E1 1144.925,E2 1144.925} C_VEL
LIN {X 0,Y 599.421,Z 549.53,A -85,B 0,C 180,E1 1149.362,E2 1149.362} C_VEL
LIN {X 0,Y 599.538,Z 549.53,A -85,B 0,C 180,E1 1153.926,E2 1153.926} C_VEL
LIN {X 0,Y 599.616,Z 549.53,A -85,B 0,C 180,E1 1158.384,E2 1158.384} C_VEL
LIN {X 0,Y 599.715,Z 549.53,A -85,B 0,C 180,E1 1162.771,E2 1162.771} C_VEL
LIN {X 0,Y 599.867,Z 549.53,A -85,B 0,C 180,E1 1167.115,E2 1167.115} C_VEL
LIN {X 0,Y 599.744,Z 550.011,A -85,B 0,C 180,E1 1170.62,E2 1170.62} C_VEL
LIN {X 0,Y 601.24,Z 561.434,A -85,B 0,C 180,E1 1170.861,E2 1170.861} C_VEL
LIN {X 0,Y 601.058,Z 599.649,A -85,B 0,C 180,E1 1171.842,E2 1171.842} C_VEL
LIN {X 0,Y 600.849,Z 634.576,A -85,B 0,C 180,E1 1173.328,E2 1173.328} C_VEL
LIN {X 0,Y 600.615,Z 668.529,A -85,B 0,C 180,E1 1175.405,E2 1175.405} C_VEL
LIN {X 0,Y 600.398,Z 698.834,A -85,B 0,C 180,E1 1177.945,E2 1177.945} C_VEL
LIN {X 0,Y 600.231,Z 724.155,A -85,B 0,C 180,E1 1180.774,E2 1180.774} C_VEL
LIN {X 0,Y 600.064,Z 745.684,A -85,B 0,C 180,E1 1184.006,E2 1184.006} C_VEL
LIN {X 0,Y 600.049,Z 760.883,A -85,B 0,C 180,E1 1187.216,E2 1187.216} C_VEL
LIN {X 0,Y 599.966,Z 771.371,A -85,B 0,C 180,E1 1190.616,E2 1190.616} C_VEL
LIN {X 0,Y 599.917,Z 776.448,A -85,B 0,C 180,E1 1193.731,E2 1193.731} C_VEL
LIN {X 0,Y 599.865,Z 777.283,A -85,B 0,C 180,E1 1196.923,E2 1196.923} C_VEL
LIN {X 0,Y 599.941,Z 773.63,A -85,B 0,C 180,E1 1200.201,E2 1200.201} C_VEL
LIN {X 0,Y 600.004,Z 763.621,A -85,B 0,C 180,E1 1203.948,E2 1203.948} C_VEL
LIN {X 0,Y 600.086,Z 748.658,A -85,B 0,C 180,E1 1207.346,E2 1207.346} C_VEL
LIN {X 0,Y 600.2,Z 728.641,A -85,B 0,C 180,E1 1210.542,E2 1210.542} C_VEL
LIN {X 0,Y 600.333,Z 703.168,A -85,B 0,C 180,E1 1213.538,E2 1213.538} C_VEL
LIN {X 0,Y 600.584,Z 673.957,A -85,B 0,C 180,E1 1216.1,E2 1216.1} C_VEL
LIN {X 0,Y 600.796,Z 641.242,A -85,B 0,C 180,E1 1218.232,E2 1218.232} C_VEL
LIN {X 0,Y 601.078,Z 604.597,A -85,B 0,C 180,E1 1219.891,E2 1219.891} C_VEL
LIN {X 0,Y 601.233,Z 567.819,A -85,B 0,C 180,E1 1220.923,E2 1220.923} C_VEL
LIN {X 0,Y 600.292,Z 551.468,A -85,B 0,C 180,E1 1221.245,E2 1221.245} C_VEL
LIN {X 0,Y 599.991,Z 549.53,A -85,B 0,C 180,E1 1221.345,E2 1221.345} C_VEL
LIN {X 0,Y 599.322,Z 549.53,A -85,B 0,C 180,E1 1226.386,E2 1226.386} C_VEL
LIN {X 0,Y 599.416,Z 549.53,A -85,B 0,C 180,E1 1231.445,E2 1231.445} C_VEL
LIN {X 0,Y 599.467,Z 549.53,A -85,B 0,C 180,E1 1236.268,E2 1236.268} C_VEL
LIN {X 0,Y 599.775,Z 549.53,A -85,B 0,C 180,E1 1240.926,E2 1240.926} C_VEL
LIN {X 0,Y 599.376,Z 549.53,A -85,B 0,C 180,E1 1245.434,E2 1245.434} C_VEL
LIN {X 0,Y 599.788,Z 549.53,A -85,B 0,C 180,E1 1249.871,E2 1249.871} C_VEL
LIN {X 0,Y 600.009,Z 549.53,A -85,B 0,C 180,E1 1254.24,E2 1254.24} C_VEL
LIN {X 0,Y 599.79,Z 549.53,A -85,B 0,C 180,E1 1259.261,E2 1259.261} C_VEL
LIN {X 0,Y 595.625,Z 549.53,A -85,B 0,C 180,E1 1260.891,E2 1260.891} C_VEL
LIN {X 0,Y 591.81,Z 549.53,A -85,B 0,C 180,E1 1262.544,E2 1262.544} C_VEL
LIN {X 0,Y 591.909,Z 549.53,A -85,B 0,C 180,E1 1268.809,E2 1268.809} C_VEL
LIN {X 0,Y 591.694,Z 549.53,A -85,B 0,C 180,E1 1274.279,E2 1274.279} C_VEL
LIN {X 0,Y 591.721,Z 549.53,A -85,B 0,C 180,E1 1279.37,E2 1279.37} C_VEL
LIN {X 0,Y 591.63,Z 549.53,A -85,B 0,C 180,E1 1284.093,E2 1284.093} C_VEL
LIN {X 0,Y 591.679,Z 549.53,A -85,B 0,C 180,E1 1288.991,E2 1288.991} C_VEL
LIN {X 0,Y 591.903,Z 549.53,A -85,B 0,C 180,E1 1294.122,E2 1294.122} C_VEL
LIN {X 0,Y 591.585,Z 549.53,A -85,B 0,C 180,E1 1300.073,E2 1300.073} C_VEL
LIN {X 0,Y 591.417,Z 549.53,A -85,B 0,C 180,E1 1305.6,E2 1305.6} C_VEL
LIN {X 0,Y 591.569,Z 549.53,A -85,B 0,C 180,E1 1310.38,E2 1310.38} C_VEL
LIN {X 0,Y 591.892,Z 549.53,A -85,B 0,C 180,E1 1315.884,E2 1315.884} C_VEL
LIN {X 0,Y 591.873,Z 549.794,A -85,B 0,C 180,E1 1319.533,E2 1319.533} C_VEL
LIN {X 0,Y 594.542,Z 558.565,A -85,B 0,C 180,E1 1319.805,E2 1319.805} C_VEL
LIN {X 0,Y 594.682,Z 624.001,A -85,B 0,C 180,E1 1320.843,E2 1320.843} C_VEL
LIN {X 0,Y 594.364,Z 663.514,A -85,B 0,C 180,E1 1322.091,E2 1322.091} C_VEL
LIN {X 0,Y 593.89,Z 701.204,A -85,B 0,C 180,E1 1323.904,E2 1323.904} C_VEL
LIN {X 0,Y 593.301,Z 737.046,A -85,B 0,C 180,E1 1326.295,E2 1326.295} C_VEL
LIN {X 0,Y 592.862,Z 768.963,A -85,B 0,C 180,E1 1329.125,E2 1329.125} C_VEL
LIN {X 0,Y 592.534,Z 795.71,A -85,B 0,C 180,E1 1332.207,E2 1332.207} C_VEL
LIN {X 0,Y 592.212,Z 817.833,A -85,B 0,C 180,E1 1335.526,E2 1335.526} C_VEL
LIN {X 0,Y 592.082,Z 836.164,A -85,B 0,C 180,E1 1339.267,E2 1339.267} C_VEL
LIN {X 0,Y 591.991,Z 847.68,A -85,B 0,C 180,E1 1342.679,E2 1342.679} C_VEL
LIN {X 0,Y 591.885,Z 853.958,A -85,B 0,C 180,E1 1345.615,E2 1345.615} C_VEL
LIN {X 0,Y 591.91,Z 857.087,A -85,B 0,C 180,E1 1348.54,E2 1348.54} C_VEL
LIN {X 0,Y 592.073,Z 857.085,A -85,B 0,C 180,E1 1351.462,E2 1351.462} C_VEL
LIN {X 0,Y 592.065,Z 852.755,A -85,B 0,C 180,E1 1355.119,E2 1355.119} C_VEL
LIN {X 0,Y 592.094,Z 842.069,A -85,B 0,C 180,E1 1359.167,E2 1359.167} C_VEL
LIN {X 0,Y 592.189,Z 826.444,A -85,B 0,C 180,E1 1362.884,E2 1362.884} C_VEL
LIN {X 0,Y 592.335,Z 804.948,A -85,B 0,C 180,E1 1366.522,E2 1366.522} C_VEL
LIN {X 0,Y 592.673,Z 779.006,A -85,B 0,C 180,E1 1369.811,E2 1369.811} C_VEL
LIN {X 0,Y 593.122,Z 748.746,A -85,B 0,C 180,E1 1372.755,E2 1372.755} C_VEL
LIN {X 0,Y 593.653,Z 714.729,A -85,B 0,C 180,E1 1375.277,E2 1375.277} C_VEL
LIN {X 0,Y 594.205,Z 677.609,A -85,B 0,C 180,E1 1377.304,E2 1377.304} C_VEL
LIN {X 0,Y 594.577,Z 638.802,A -85,B 0,C 180,E1 1378.76,E2 1378.76} C_VEL
LIN {X 0,Y 594.881,Z 600.976,A -85,B 0,C 180,E1 1379.589,E2 1379.589} C_VEL
LIN {X 0,Y 593.84,Z 554.965,A -85,B 0,C 180,E1 1380.284,E2 1380.284} C_VEL
LIN {X 0,Y 591.866,Z 549.53,A -85,B 0,C 180,E1 1380.471,E2 1380.471} C_VEL
LIN {X 0,Y 591.743,Z 549.53,A -85,B 0,C 180,E1 1385.912,E2 1385.912} C_VEL
LIN {X 0,Y 591.478,Z 549.53,A -85,B 0,C 180,E1 1391.556,E2 1391.556} C_VEL
LIN {X 0,Y 591.633,Z 549.53,A -85,B 0,C 180,E1 1396.472,E2 1396.472} C_VEL
LIN {X 0,Y 591.686,Z 549.53,A -85,B 0,C 180,E1 1402.255,E2 1402.255} C_VEL
LIN {X 0,Y 591.441,Z 549.53,A -85,B 0,C 180,E1 1407.596,E2 1407.596} C_VEL
LIN {X 0,Y 591.519,Z 549.53,A -85,B 0,C 180,E1 1412.658,E2 1412.658} C_VEL
LIN {X 0,Y 591.501,Z 549.53,A -85,B 0,C 180,E1 1417.493,E2 1417.493} C_VEL
LIN {X 0,Y 591.778,Z 549.53,A -85,B 0,C 180,E1 1422.174,E2 1422.174} C_VEL
LIN {X 0,Y 591.607,Z 549.53,A -85,B 0,C 180,E1 1428.216,E2 1428.216} C_VEL
LIN {X 0,Y 592.07,Z 549.53,A -85,B 0,C 180,E1 1434.138,E2 1434.138} C_VEL
LIN {X 0,Y 591.8,Z 549.53,A -85,B 0,C 180,E1 1439.988,E2 1439.988} C_VEL
LIN {X 0,Y 591.84,Z 549.53,A -85,B 0,C 180,E1 1444.374,E2 1444.374} C_VEL
LIN {X 0,Y 591.895,Z 549.53,A -85,B 0,C 180,E1 1448.785,E2 1448.785} C_VEL
LIN {X 0,Y 591.686,Z 549.53,A -85,B 0,C 180,E1 1454.267,E2 1454.267} C_VEL
LIN {X 0,Y 591.712,Z 549.53,A -85,B 0,C 180,E1 1459.344,E2 1459.344} C_VEL
LIN {X 0,Y 591.625,Z 549.53,A -85,B 0,C 180,E1 1464.066,E2 1464.066} C_VEL
LIN {X 0,Y 591.648,Z 549.53,A -85,B 0,C 180,E1 1468.965,E2 1468.965} C_VEL
LIN {X 0,Y 591.89,Z 549.53,A -85,B 0,C 180,E1 1474.093,E2 1474.093} C_VEL
LIN {X 0,Y 591.608,Z 549.53,A -85,B 0,C 180,E1 1480.073,E2 1480.073} C_VEL
LIN {X 0,Y 591.418,Z 549.53,A -85,B 0,C 180,E1 1485.565,E2 1485.565} C_VEL
LIN {X 0,Y 591.581,Z 549.53,A -85,B 0,C 180,E1 1490.378,E2 1490.378} C_VEL
LIN {X 0,Y 591.864,Z 549.53,A -85,B 0,C 180,E1 1495.88,E2 1495.88} C_VEL
LIN {X 0,Y 591.68,Z 549.53,A -85,B 0,C 180,E1 1501.014,E2 1501.014} C_VEL
LIN {X 0,Y 591.659,Z 549.53,A -85,B 0,C 180,E1 1507.506,E2 1507.506} C_VEL
LIN {X 0,Y 591.884,Z 549.53,A -85,B 0,C 180,E1 1512.184,E2 1512.184} C_VEL
LIN {X 0,Y 591.73,Z 549.53,A -85,B 0,C 180,E1 1518.227,E2 1518.227} C_VEL
LIN {X 0,Y 591.833,Z 549.53,A -85,B 0,C 180,E1 1522.675,E2 1522.675} C_VEL
LIN {X 0,Y 591.96,Z 549.53,A -85,B 0,C 180,E1 1527.076,E2 1527.076} C_VEL
LIN {X 0,Y 591.767,Z 549.53,A -85,B 0,C 180,E1 1530.227,E2 1530.227} C_VEL
LIN {X 0,Y 594.053,Z 559.065,A -85,B 0,C 180,E1 1530.499,E2 1530.499} C_VEL
LIN {X 0,Y 593.909,Z 597.458,A -85,B 0,C 180,E1 1531.455,E2 1531.455} C_VEL
LIN {X 0,Y 593.5,Z 634.059,A -85,B 0,C 180,E1 1533.005,E2 1533.005} C_VEL
LIN {X 0,Y 593.111,Z 666.89,A -85,B 0,C 180,E1 1535.016,E2 1535.016} C_VEL
LIN {X 0,Y 592.747,Z 696.755,A -85,B 0,C 180,E1 1537.496,E2 1537.496} C_VEL
LIN {X 0,Y 592.47,Z 722.933,A -85,B 0,C 180,E1 1540.412,E2 1540.412} C_VEL
LIN {X 0,Y 592.24,Z 744.128,A -85,B 0,C 180,E1 1543.577,E2 1543.577} C_VEL
LIN {X 0,Y 592.182,Z 760.828,A -85,B 0,C 180,E1 1547.084,E2 1547.084} C_VEL
LIN {X 0,Y 592.127,Z 770.45,A -85,B 0,C 180,E1 1550.157,E2 1550.157} C_VEL
LIN {X 0,Y 592.012,Z 776.196,A -85,B 0,C 180,E1 1553.481,E2 1553.481} C_VEL
LIN {X 0,Y 591.967,Z 777.083,A -85,B 0,C 180,E1 1557.312,E2 1557.312} C_VEL
LIN {X 0,Y 592.097,Z 772.894,A -85,B 0,C 180,E1 1560.644,E2 1560.644} C_VEL
LIN {X 0,Y 592.113,Z 763.454,A -85,B 0,C 180,E1 1564.101,E2 1564.101} C_VEL
LIN {X 0,Y 592.215,Z 749.462,A -85,B 0,C 180,E1 1567.347,E2 1567.347} C_VEL
LIN {X 0,Y 592.407,Z 729.483,A -85,B 0,C 180,E1 1570.619,E2 1570.619} C_VEL
LIN {X 0,Y 592.641,Z 704.068,A -85,B 0,C 180,E1 1573.684,E2 1573.684} C_VEL
LIN {X 0,Y 593.007,Z 674.322,A -85,B 0,C 180,E1 1576.341,E2 1576.341} C_VEL
LIN {X 0,Y 593.402,Z 641.063,A -85,B 0,C 180,E1 1578.535,E2 1578.535} C_VEL
LIN {X 0,Y 593.824,Z 604.849,A -85,B 0,C 180,E1 1580.193,E2 1580.193} C_VEL
LIN {X 0,Y 594.042,Z 569.619,A -85,B 0,C 180,E1 1581.209,E2 1581.209} C_VEL
LIN {X 0,Y 593.365,Z 553.919,A -85,B 0,C 180,E1 1581.523,E2 1581.523} C_VEL
LIN {X 0,Y 592.013,Z 549.53,A -85,B 0,C 180,E1 1581.703,E2 1581.703} C_VEL
LIN {X 0,Y 591.435,Z 549.53,A -85,B 0,C 180,E1 1587.625,E2 1587.625} C_VEL
LIN {X 0,Y 591.533,Z 549.53,A -85,B 0,C 180,E1 1592.686,E2 1592.686} C_VEL
LIN {X 0,Y 591.49,Z 549.53,A -85,B 0,C 180,E1 1597.519,E2 1597.519} C_VEL
LIN {X 0,Y 591.865,Z 549.53,A -85,B 0,C 180,E1 1602.202,E2 1602.202} C_VEL
LIN {X 0,Y 591.59,Z 549.53,A -85,B 0,C 180,E1 1608.241,E2 1608.241} C_VEL
LIN {X 0,Y 592.076,Z 549.53,A -85,B 0,C 180,E1 1614.162,E2 1614.162} C_VEL
LIN {X 0,Y 591.797,Z 549.53,A -85,B 0,C 180,E1 1620.012,E2 1620.012} C_VEL
LIN {X 0,Y 591.81,Z 549.53,A -85,B 0,C 180,E1 1622.544,E2 1622.544} C_VEL
LIN {X 0,Y 589.375,Z 549.53,A -85,B 0,C 180,E1 1623.793,E2 1623.793} C_VEL
LIN {X 0,Y 583.893,Z 549.53,A -85,B 0,C 180,E1 1625.663,E2 1625.663} C_VEL
LIN {X 0,Y 583.803,Z 549.53,A -85,B 0,C 180,E1 1625.879,E2 1625.879} C_VEL
LIN {X 0,Y 583.763,Z 549.53,A -85,B 0,C 180,E1 1630.805,E2 1630.805} C_VEL
LIN {X 0,Y 583.717,Z 549.53,A -85,B 0,C 180,E1 1634.991,E2 1634.991} C_VEL
LIN {X 0,Y 583.778,Z 549.53,A -85,B 0,C 180,E1 1639.644,E2 1639.644} C_VEL
LIN {X 0,Y 583.671,Z 549.53,A -85,B 0,C 180,E1 1644.442,E2 1644.442} C_VEL
LIN {X 0,Y 583.698,Z 549.53,A -85,B 0,C 180,E1 1649.426,E2 1649.426} C_VEL
LIN {X 0,Y 583.913,Z 549.53,A -85,B 0,C 180,E1 1654.655,E2 1654.655} C_VEL
LIN {X 0,Y 583.667,Z 549.53,A -85,B 0,C 180,E1 1660.272,E2 1660.272} C_VEL
LIN {X 0,Y 583.606,Z 549.53,A -85,B 0,C 180,E1 1666.388,E2 1666.388} C_VEL
LIN {X 0,Y 583.721,Z 549.53,A -85,B 0,C 180,E1 1671.653,E2 1671.653} C_VEL
LIN {X 0,Y 583.95,Z 549.53,A -85,B 0,C 180,E1 1677.136,E2 1677.136} C_VEL
LIN {X 0,Y 583.921,Z 549.53,A -85,B 0,C 180,E1 1679.046,E2 1679.046} C_VEL
LIN {X 0,Y 587.702,Z 559.136,A -85,B 0,C 180,E1 1679.424,E2 1679.424} C_VEL
LIN {X 0,Y 587.805,Z 623.673,A -85,B 0,C 180,E1 1680.461,E2 1680.461} C_VEL
LIN {X 0,Y 587.313,Z 662.712,A -85,B 0,C 180,E1 1681.692,E2 1681.692} C_VEL
LIN {X 0,Y 586.64,Z 700.7,A -85,B 0,C 180,E1 1683.526,E2 1683.526} C_VEL
LIN {X 0,Y 585.894,Z 737.048,A -85,B 0,C 180,E1 1685.976,E2 1685.976} C_VEL
LIN {X 0,Y 585.256,Z 768.962,A -85,B 0,C 180,E1 1688.841,E2 1688.841} C_VEL
LIN {X 0,Y 584.75,Z 795.712,A -85,B 0,C 180,E1 1691.962,E2 1691.962} C_VEL
LIN {X 0,Y 584.373,Z 818.568,A -85,B 0,C 180,E1 1695.456,E2 1695.456} C_VEL
LIN {X 0,Y 584.228,Z 836.848,A -85,B 0,C 180,E1 1699.288,E2 1699.288} C_VEL
LIN {X 0,Y 584.143,Z 849.023,A -85,B 0,C 180,E1 1703.102,E2 1703.102} C_VEL
LIN {X 0,Y 584.084,Z 855.908,A -85,B 0,C 180,E1 1707.039,E2 1707.039} C_VEL
LIN {X 0,Y 584.051,Z 857.5,A -85,B 0,C 180,E1 1710.001,E2 1710.001} C_VEL
LIN {X 0,Y 584.03,Z 855.905,A -85,B 0,C 180,E1 1712.963,E2 1712.963} C_VEL
LIN {X 0,Y 584.087,Z 850.432,A -85,B 0,C 180,E1 1716.31,E2 1716.31} C_VEL
LIN {X 0,Y 584.071,Z 839.392,A -85,B 0,C 180,E1 1720.044,E2 1720.044} C_VEL
LIN {X 0,Y 584.313,Z 823.097,A -85,B 0,C 180,E1 1723.711,E2 1723.711} C_VEL
LIN {X 0,Y 584.592,Z 801.55,A -85,B 0,C 180,E1 1727.24,E2 1727.24} C_VEL
LIN {X 0,Y 585.124,Z 774.603,A -85,B 0,C 180,E1 1730.573,E2 1730.573} C_VEL
LIN {X 0,Y 585.783,Z 742.732,A -85,B 0,C 180,E1 1733.569,E2 1733.569} C_VEL
LIN {X 0,Y 586.439,Z 708.068,A -85,B 0,C 180,E1 1736.034,E2 1736.034} C_VEL
LIN {X 0,Y 587.149,Z 670.776,A -85,B 0,C 180,E1 1737.968,E2 1737.968} C_VEL
LIN {X 0,Y 587.64,Z 633.262,A -85,B 0,C 180,E1 1739.291,E2 1739.291} C_VEL
LIN {X 0,Y 587.972,Z 591.059,A -85,B 0,C 180,E1 1740.118,E2 1740.118} C_VEL
LIN {X 0,Y 587.013,Z 557.786,A -85,B 0,C 180,E1 1740.635,E2 1740.635} C_VEL
LIN {X 0,Y 583.841,Z 549.53,A -85,B 0,C 180,E1 1740.966,E2 1740.966} C_VEL
LIN {X 0,Y 583.817,Z 549.53,A -85,B 0,C 180,E1 1746.746,E2 1746.746} C_VEL
LIN {X 0,Y 583.573,Z 549.53,A -85,B 0,C 180,E1 1752.247,E2 1752.247} C_VEL
LIN {X 0,Y 583.735,Z 549.53,A -85,B 0,C 180,E1 1757.764,E2 1757.764} C_VEL
LIN {X 0,Y 583.73,Z 549.53,A -85,B 0,C 180,E1 1763.512,E2 1763.512} C_VEL
LIN {X 0,Y 583.642,Z 549.53,A -85,B 0,C 180,E1 1768.856,E2 1768.856} C_VEL
LIN {X 0,Y 583.789,Z 549.53,A -85,B 0,C 180,E1 1774.786,E2 1774.786} C_VEL
LIN {X 0,Y 583.892,Z 549.53,A -85,B 0,C 180,E1 1780.36,E2 1780.36} C_VEL
LIN {X 0,Y 583.648,Z 549.53,A -85,B 0,C 180,E1 1785.007,E2 1785.007} C_VEL
LIN {X 0,Y 583.93,Z 549.53,A -85,B 0,C 180,E1 1789.568,E2 1789.568} C_VEL
LIN {X 0,Y 584.153,Z 549.53,A -85,B 0,C 180,E1 1794.058,E2 1794.058} C_VEL
LIN {X 0,Y 583.922,Z 549.53,A -85,B 0,C 180,E1 1799.988,E2 1799.988} C_VEL
LIN {X 0,Y 583.94,Z 549.53,A -85,B 0,C 180,E1 1804.433,E2 1804.433} C_VEL
LIN {X 0,Y 583.959,Z 549.53,A -85,B 0,C 180,E1 1808.905,E2 1808.905} C_VEL
LIN {X 0,Y 584.015,Z 549.53,A -85,B 0,C 180,E1 1813.431,E2 1813.431} C_VEL
LIN {X 0,Y 583.937,Z 549.53,A -85,B 0,C 180,E1 1818.048,E2 1818.048} C_VEL
LIN {X 0,Y 583.83,Z 549.53,A -85,B 0,C 180,E1 1822.793,E2 1822.793} C_VEL
LIN {X 0,Y 583.713,Z 549.53,A -85,B 0,C 180,E1 1828.48,E2 1828.48} C_VEL
LIN {X 0,Y 583.93,Z 549.53,A -85,B 0,C 180,E1 1834.624,E2 1834.624} C_VEL
LIN {X 0,Y 583.725,Z 549.53,A -85,B 0,C 180,E1 1840.235,E2 1840.235} C_VEL
LIN {X 0,Y 583.613,Z 549.53,A -85,B 0,C 180,E1 1846.352,E2 1846.352} C_VEL
LIN {X 0,Y 583.715,Z 549.53,A -85,B 0,C 180,E1 1851.65,E2 1851.65} C_VEL
LIN {X 0,Y 583.876,Z 549.53,A -85,B 0,C 180,E1 1857.128,E2 1857.128} C_VEL
LIN {X 0,Y 583.683,Z 549.53,A -85,B 0,C 180,E1 1862.265,E2 1862.265} C_VEL
LIN {X 0,Y 583.763,Z 549.53,A -85,B 0,C 180,E1 1867.184,E2 1867.184} C_VEL
LIN {X 0,Y 583.856,Z 549.53,A -85,B 0,C 180,E1 1872.911,E2 1872.911} C_VEL
LIN {X 0,Y 583.852,Z 549.53,A -85,B 0,C 180,E1 1878.066,E2 1878.066} C_VEL
LIN {X 0,Y 583.926,Z 549.53,A -85,B 0,C 180,E1 1882.575,E2 1882.575} C_VEL
LIN {X 0,Y 584.062,Z 549.53,A -85,B 0,C 180,E1 1887.037,E2 1887.037} C_VEL
LIN {X 0,Y 583.817,Z 549.53,A -85,B 0,C 180,E1 1889.86,E2 1889.86} C_VEL
LIN {X 0,Y 586.929,Z 560.033,A -85,B 0,C 180,E1 1890.183,E2 1890.183} C_VEL
LIN {X 0,Y 586.686,Z 597.933,A -85,B 0,C 180,E1 1891.15,E2 1891.15} C_VEL
LIN {X 0,Y 586.196,Z 633.52,A -85,B 0,C 180,E1 1892.673,E2 1892.673} C_VEL
LIN {X 0,Y 585.62,Z 666.541,A -85,B 0,C 180,E1 1894.71,E2 1894.71} C_VEL
LIN {X 0,Y 585.069,Z 696.88,A -85,B 0,C 180,E1 1897.257,E2 1897.257} C_VEL
LIN {X 0,Y 584.683,Z 723.084,A -85,B 0,C 180,E1 1900.219,E2 1900.219} C_VEL
LIN {X 0,Y 584.396,Z 744.292,A -85,B 0,C 180,E1 1903.437,E2 1903.437} C_VEL
LIN {X 0,Y 584.279,Z 760.446,A -85,B 0,C 180,E1 1906.864,E2 1906.864} C_VEL
LIN {X 0,Y 584.22,Z 771.234,A -85,B 0,C 180,E1 1910.407,E2 1910.407} C_VEL
LIN {X 0,Y 584.051,Z 775.461,A -85,B 0,C 180,E1 1912.801,E2 1912.801} C_VEL
LIN {X 0,Y 584.006,Z 777.485,A -85,B 0,C 180,E1 1916.056,E2 1916.056} C_VEL
LIN {X 0,Y 584.083,Z 775.107,A -85,B 0,C 180,E1 1919.397,E2 1919.397} C_VEL
LIN {X 0,Y 584.081,Z 767.778,A -85,B 0,C 180,E1 1922.856,E2 1922.856} C_VEL
LIN {X 0,Y 584.219,Z 754.545,A -85,B 0,C 180,E1 1926.446,E2 1926.446} C_VEL
LIN {X 0,Y 584.416,Z 737.011,A -85,B 0,C 180,E1 1929.694,E2 1929.694} C_VEL
LIN {X 0,Y 584.731,Z 714.103,A -85,B 0,C 180,E1 1932.808,E2 1932.808} C_VEL
LIN {X 0,Y 585.268,Z 685.611,A -85,B 0,C 180,E1 1935.686,E2 1935.686} C_VEL
LIN {X 0,Y 585.798,Z 655.141,A -85,B 0,C 180,E1 1937.98,E2 1937.98} C_VEL
LIN {X 0,Y 586.402,Z 621.004,A -85,B 0,C 180,E1 1939.845,E2 1939.845} C_VEL
LIN {X 0,Y 586.789,Z 584.353,A -85,B 0,C 180,E1 1941.182,E2 1941.182} C_VEL
LIN {X 0,Y 586.182,Z 556.291,A -85,B 0,C 180,E1 1941.822,E2 1941.822} C_VEL
LIN {X 0,Y 584.07,Z 549.53,A -85,B 0,C 180,E1 1942.11,E2 1942.11} C_VEL
LIN {X 0,Y 583.605,Z 549.53,A -85,B 0,C 180,E1 1948.567,E2 1948.567} C_VEL
LIN {X 0,Y 583.777,Z 549.53,A -85,B 0,C 180,E1 1954.783,E2 1954.783} C_VEL
LIN {X 0,Y 583.945,Z 549.53,A -85,B 0,C 180,E1 1960.388,E2 1960.388} C_VEL
LIN {X 0,Y 583.616,Z 549.53,A -85,B 0,C 180,E1 1965.032,E2 1965.032} C_VEL
LIN {X 0,Y 583.766,Z 549.53,A -85,B 0,C 180,E1 1971.092,E2 1971.092} C_VEL
LIN {X 0,Y 583.867,Z 549.53,A -85,B 0,C 180,E1 1975.566,E2 1975.566} C_VEL
LIN {X 0,Y 583.918,Z 549.53,A -85,B 0,C 180,E1 1980.012,E2 1980.012} C_VEL
LIN {X 0,Y 583.941,Z 549.53,A -85,B 0,C 180,E1 1984.458,E2 1984.458} C_VEL
LIN {X 0,Y 583.803,Z 549.53,A -85,B 0,C 180,E1 1985.879,E2 1985.879} C_VEL
LIN {X 0,Y 580.019,Z 549.53,A -85,B 0,C 180,E1 1987.557,E2 1987.557} C_VEL
LIN {X 0,Y 576.003,Z 549.53,A -85,B 0,C 180,E1 1989.258,E2 1989.258} C_VEL
LIN {X 0,Y 575.946,Z 549.53,A -85,B 0,C 180,E1 1994.21,E2 1994.21} C_VEL
LIN {X 0,Y 575.863,Z 549.53,A -85,B 0,C 180,E1 1999.925,E2 1999.925} C_VEL
LIN {X 0,Y 575.744,Z 549.53,A -85,B 0,C 180,E1 2004.801,E2 2004.801} C_VEL
LIN {X 0,Y 575.742,Z 549.53,A -85,B 0,C 180,E1 2010.128,E2 2010.128} C_VEL
LIN {X 0,Y 575.91,Z 549.53,A -85,B 0,C 180,E1 2015.207,E2 2015.207} C_VEL
LIN {X 0,Y 575.755,Z 549.53,A -85,B 0,C 180,E1 2020.942,E2 2020.942} C_VEL
LIN {X 0,Y 575.768,Z 549.53,A -85,B 0,C 180,E1 2027.213,E2 2027.213} C_VEL
LIN {X 0,Y 575.87,Z 549.53,A -85,B 0,C 180,E1 2032.938,E2 2032.938} C_VEL
LIN {X 0,Y 576.019,Z 549.53,A -85,B 0,C 180,E1 2038.58,E2 2038.58} C_VEL
LIN {X 0,Y 580.945,Z 564.068,A -85,B 0,C 180,E1 2039.099,E2 2039.099} C_VEL
LIN {X 0,Y 580.891,Z 624.62,A -85,B 0,C 180,E1 2040.098,E2 2040.098} C_VEL
LIN {X 0,Y 580.254,Z 663.605,A -85,B 0,C 180,E1 2041.354,E2 2041.354} C_VEL
LIN {X 0,Y 579.376,Z 702.128,A -85,B 0,C 180,E1 2043.256,E2 2043.256} C_VEL
LIN {X 0,Y 578.462,Z 736.879,A -85,B 0,C 180,E1 2045.634,E2 2045.634} C_VEL
LIN {X 0,Y 577.636,Z 768.962,A -85,B 0,C 180,E1 2048.548,E2 2048.548} C_VEL
LIN {X 0,Y 577.019,Z 795.713,A -85,B 0,C 180,E1 2051.711,E2 2051.711} C_VEL
LIN {X 0,Y 576.56,Z 818.566,A -85,B 0,C 180,E1 2055.254,E2 2055.254} C_VEL
LIN {X 0,Y 576.349,Z 836.848,A -85,B 0,C 180,E1 2059.14,E2 2059.14} C_VEL
LIN {X 0,Y 576.2,Z 847.68,A -85,B 0,C 180,E1 2062.477,E2 2062.477} C_VEL
LIN {X 0,Y 576.1,Z 853.958,A -85,B 0,C 180,E1 2065.494,E2 2065.494} C_VEL
LIN {X 0,Y 576.133,Z 857.087,A -85,B 0,C 180,E1 2068.5,E2 2068.5} C_VEL
LIN {X 0,Y 576.278,Z 857.086,A -85,B 0,C 180,E1 2071.502,E2 2071.502} C_VEL
LIN {X 0,Y 576.257,Z 851.88,A -85,B 0,C 180,E1 2075.692,E2 2075.692} C_VEL
LIN {X 0,Y 576.281,Z 842.068,A -85,B 0,C 180,E1 2079.42,E2 2079.42} C_VEL
LIN {X 0,Y 576.455,Z 826.442,A -85,B 0,C 180,E1 2083.242,E2 2083.242} C_VEL
LIN {X 0,Y 576.775,Z 805.394,A -85,B 0,C 180,E1 2086.915,E2 2086.915} C_VEL
LIN {X 0,Y 577.384,Z 779.858,A -85,B 0,C 180,E1 2090.262,E2 2090.262} C_VEL
LIN {X 0,Y 578.127,Z 749.618,A -85,B 0,C 180,E1 2093.302,E2 2093.302} C_VEL
LIN {X 0,Y 579.025,Z 715.713,A -85,B 0,C 180,E1 2095.895,E2 2095.895} C_VEL
LIN {X 0,Y 579.918,Z 679.727,A -85,B 0,C 180,E1 2097.93,E2 2097.93} C_VEL
LIN {X 0,Y 580.633,Z 642.49,A -85,B 0,C 180,E1 2099.398,E2 2099.398} C_VEL
LIN {X 0,Y 581.114,Z 605.875,A -85,B 0,C 180,E1 2100.281,E2 2100.281} C_VEL
LIN {X 0,Y 580.314,Z 560.516,A -85,B 0,C 180,E1 2100.989,E2 2100.989} C_VEL
LIN {X 0,Y 575.803,Z 549.53,A -85,B 0,C 180,E1 2101.497,E2 2101.497} C_VEL
LIN {X 0,Y 575.907,Z 549.53,A -85,B 0,C 180,E1 2107.062,E2 2107.062} C_VEL
LIN {X 0,Y 575.686,Z 549.53,A -85,B 0,C 180,E1 2112.964,E2 2112.964} C_VEL
LIN {X 0,Y 575.774,Z 549.53,A -85,B 0,C 180,E1 2119.06,E2 2119.06} C_VEL
LIN {X 0,Y 575.686,Z 549.53,A -85,B 0,C 180,E1 2124.777,E2 2124.777} C_VEL
LIN {X 0,Y 575.721,Z 549.53,A -85,B 0,C 180,E1 2130.125,E2 2130.125} C_VEL
LIN {X 0,Y 575.855,Z 549.53,A -85,B 0,C 180,E1 2135.204,E2 2135.204} C_VEL
LIN {X 0,Y 575.963,Z 549.53,A -85,B 0,C 180,E1 2140.598,E2 2140.598} C_VEL
LIN {X 0,Y 575.791,Z 549.53,A -85,B 0,C 180,E1 2144.797,E2 2144.797} C_VEL
LIN {X 0,Y 575.878,Z 549.53,A -85,B 0,C 180,E1 2150.944,E2 2150.944} C_VEL
LIN {X 0,Y 575.963,Z 549.53,A -85,B 0,C 180,E1 2155.48,E2 2155.48} C_VEL
LIN {X 0,Y 576.021,Z 549.53,A -85,B 0,C 180,E1 2159.988,E2 2159.988} C_VEL
LIN {X 0,Y 576.025,Z 549.53,A -85,B 0,C 180,E1 2164.494,E2 2164.494} C_VEL
LIN {X 0,Y 576.039,Z 549.53,A -85,B 0,C 180,E1 2169.028,E2 2169.028} C_VEL
LIN {X 0,Y 575.942,Z 549.53,A -85,B 0,C 180,E1 2174.199,E2 2174.199} C_VEL
LIN {X 0,Y 575.85,Z 549.53,A -85,B 0,C 180,E1 2179.899,E2 2179.899} C_VEL
LIN {X 0,Y 575.74,Z 549.53,A -85,B 0,C 180,E1 2184.774,E2 2184.774} C_VEL
LIN {X 0,Y 575.718,Z 549.53,A -85,B 0,C 180,E1 2190.119,E2 2190.119} C_VEL
LIN {X 0,Y 575.924,Z 549.53,A -85,B 0,C 180,E1 2195.175,E2 2195.175} C_VEL
LIN {X 0,Y 575.811,Z 549.53,A -85,B 0,C 180,E1 2200.904,E2 2200.904} C_VEL
LIN {X 0,Y 575.753,Z 549.53,A -85,B 0,C 180,E1 2207.178,E2 2207.178} C_VEL
LIN {X 0,Y 575.864,Z 549.53,A -85,B 0,C 180,E1 2212.935,E2 2212.935} C_VEL
LIN {X 0,Y 575.858,Z 549.53,A -85,B 0,C 180,E1 2218.392,E2 2218.392} C_VEL
LIN {X 0,Y 575.695,Z 549.53,A -85,B 0,C 180,E1 2223.537,E2 2223.537} C_VEL
LIN {X 0,Y 575.779,Z 549.53,A -85,B 0,C 180,E1 2228.473,E2 2228.473} C_VEL
LIN {X 0,Y 575.932,Z 549.53,A -85,B 0,C 180,E1 2233.248,E2 2233.248} C_VEL
LIN {X 0,Y 575.949,Z 549.53,A -85,B 0,C 180,E1 2237.9,E2 2237.9} C_VEL
LIN {X 0,Y 576.021,Z 549.53,A -85,B 0,C 180,E1 2242.472,E2 2242.472} C_VEL
LIN {X 0,Y 576.154,Z 549.53,A -85,B 0,C 180,E1 2246.996,E2 2246.996} C_VEL
LIN {X 0,Y 575.919,Z 549.53,A -85,B 0,C 180,E1 2249.483,E2 2249.483} C_VEL
LIN {X 0,Y 579.806,Z 563.506,A -85,B 0,C 180,E1 2249.906,E2 2249.906} C_VEL
LIN {X 0,Y 579.382,Z 601.071,A -85,B 0,C 180,E1 2250.932,E2 2250.932} C_VEL
LIN {X 0,Y 578.723,Z 636.588,A -85,B 0,C 180,E1 2252.521,E2 2252.521} C_VEL
LIN {X 0,Y 578.043,Z 670.072,A -85,B 0,C 180,E1 2254.678,E2 2254.678} C_VEL
LIN {X 0,Y 577.354,Z 700.534,A -85,B 0,C 180,E1 2257.375,E2 2257.375} C_VEL
LIN {X 0,Y 576.923,Z 725.756,A -85,B 0,C 180,E1 2260.358,E2 2260.358} C_VEL
LIN {X 0,Y 576.515,Z 747.379,A -85,B 0,C 180,E1 2263.84,E2 2263.84} C_VEL
LIN {X 0,Y 576.327,Z 763.049,A -85,B 0,C 180,E1 2267.469,E2 2267.469} C_VEL
LIN {X 0,Y 576.277,Z 771.998,A -85,B 0,C 180,E1 2270.701,E2 2270.701} C_VEL
LIN {X 0,Y 576.092,Z 776.409,A -85,B 0,C 180,E1 2273.601,E2 2273.601} C_VEL
LIN {X 0,Y 576.065,Z 777.243,A -85,B 0,C 180,E1 2277.101,E2 2277.101} C_VEL
LIN {X 0,Y 576.285,Z 772.664,A -85,B 0,C 180,E1 2280.886,E2 2280.886} C_VEL
LIN {X 0,Y 576.363,Z 763.133,A -85,B 0,C 180,E1 2284.417,E2 2284.417} C_VEL
LIN {X 0,Y 576.533,Z 747.35,A -85,B 0,C 180,E1 2288.075,E2 2288.075} C_VEL
LIN {X 0,Y 576.838,Z 726.078,A -85,B 0,C 180,E1 2291.511,E2 2291.511} C_VEL
LIN {X 0,Y 577.345,Z 700.809,A -85,B 0,C 180,E1 2294.506,E2 2294.506} C_VEL
LIN {X 0,Y 578.052,Z 670.651,A -85,B 0,C 180,E1 2297.186,E2 2297.186} C_VEL
LIN {X 0,Y 578.739,Z 637.358,A -85,B 0,C 180,E1 2299.346,E2 2299.346} C_VEL
LIN {X 0,Y 579.366,Z 601.944,A -85,B 0,C 180,E1 2300.947,E2 2300.947} C_VEL
LIN {X 0,Y 579.803,Z 566.464,A -85,B 0,C 180,E1 2301.942,E2 2301.942} C_VEL
LIN {X 0,Y 578.677,Z 557.219,A -85,B 0,C 180,E1 2302.167,E2 2302.167} C_VEL
LIN {X 0,Y 576.113,Z 549.53,A -85,B 0,C 180,E1 2302.433,E2 2302.433} C_VEL
LIN {X 0,Y 575.7,Z 549.53,A -85,B 0,C 180,E1 2308.406,E2 2308.406} C_VEL
LIN {X 0,Y 575.771,Z 549.53,A -85,B 0,C 180,E1 2313.562,E2 2313.562} C_VEL
LIN {X 0,Y 576.007,Z 549.53,A -85,B 0,C 180,E1 2320.106,E2 2320.106} C_VEL
LIN {X 0,Y 575.753,Z 549.53,A -85,B 0,C 180,E1 2324.822,E2 2324.822} C_VEL
LIN {X 0,Y 575.887,Z 549.53,A -85,B 0,C 180,E1 2330.969,E2 2330.969} C_VEL
LIN {X 0,Y 575.972,Z 549.53,A -85,B 0,C 180,E1 2335.506,E2 2335.506} C_VEL
LIN {X 0,Y 576.017,Z 549.53,A -85,B 0,C 180,E1 2340.012,E2 2340.012} C_VEL
LIN {X 0,Y 575.92,Z 549.53,A -85,B 0,C 180,E1 2345.348,E2 2345.348} C_VEL
LIN {X 0,Y 576.003,Z 549.53,A -85,B 0,C 180,E1 2349.258,E2 2349.258} C_VEL
LIN {X 0,Y 571.951,Z 549.53,A -85,B 0,C 180,E1 2350.953,E2 2350.953} C_VEL
LIN {X 0,Y 568.051,Z 549.53,A -85,B 0,C 180,E1 2352.671,E2 2352.671} C_VEL
LIN {X 0,Y 568.063,Z 549.53,A -85,B 0,C 180,E1 2358.597,E2 2358.597} C_VEL
LIN {X 0,Y 567.942,Z 549.53,A -85,B 0,C 180,E1 2363.495,E2 2363.495} C_VEL
LIN {X 0,Y 567.881,Z 549.53,A -85,B 0,C 180,E1 2368.732,E2 2368.732} C_VEL
LIN {X 0,Y 567.99,Z 549.53,A -85,B 0,C 180,E1 2374.556,E2 2374.556} C_VEL
LIN {X 0,Y 567.805,Z 549.53,A -85,B 0,C 180,E1 2379.635,E2 2379.635} C_VEL
LIN {X 0,Y 567.675,Z 549.53,A -85,B 0,C 180,E1 2385.871,E2 2385.871} C_VEL
LIN {X 0,Y 567.83,Z 549.53,A -85,B 0,C 180,E1 2390.418,E2 2390.418} C_VEL
LIN {X 0,Y 568.05,Z 549.53,A -85,B 0,C 180,E1 2396.093,E2 2396.093} C_VEL
LIN {X 0,Y 568.106,Z 549.53,A -85,B 0,C 180,E1 2398.088,E2 2398.088} C_VEL
LIN {X 0,Y 574.18,Z 564.408,A -85,B 0,C 180,E1 2398.699,E2 2398.699} C_VEL
LIN {X 0,Y 574.039,Z 624.619,A -85,B 0,C 180,E1 2399.704,E2 2399.704} C_VEL
LIN {X 0,Y 573.259,Z 663.834,A -85,B 0,C 180,E1 2400.982,E2 2400.982} C_VEL
LIN {X 0,Y 572.265,Z 700.784,A -85,B 0,C 180,E1 2402.813,E2 2402.813} C_VEL
LIN {X 0,Y 571.072,Z 736.872,A -85,B 0,C 180,E1 2405.298,E2 2405.298} C_VEL
LIN {X 0,Y 570.064,Z 768.962,A -85,B 0,C 180,E1 2408.249,E2 2408.249} C_VEL
LIN {X 0,Y 569.314,Z 795.714,A -85,B 0,C 180,E1 2411.455,E2 2411.455} C_VEL
LIN {X 0,Y 568.755,Z 818.206,A -85,B 0,C 180,E1 2414.982,E2 2414.982} C_VEL
LIN {X 0,Y 568.417,Z 834.987,A -85,B 0,C 180,E1 2418.517,E2 2418.517} C_VEL
LIN {X 0,Y 568.304,Z 847.68,A -85,B 0,C 180,E1 2422.372,E2 2422.372} C_VEL
LIN {X 0,Y 568.22,Z 853.958,A -85,B 0,C 180,E1 2425.432,E2 2425.432} C_VEL
LIN {X 0,Y 568.261,Z 857.087,A -85,B 0,C 180,E1 2428.479,E2 2428.479} C_VEL
LIN {X 0,Y 568.394,Z 857.086,A -85,B 0,C 180,E1 2431.522,E2 2431.522} C_VEL
LIN {X 0,Y 568.361,Z 852.396,A -85,B 0,C 180,E1 2435.518,E2 2435.518} C_VEL
LIN {X 0,Y 568.37,Z 842.068,A -85,B 0,C 180,E1 2439.553,E2 2439.553} C_VEL
LIN {X 0,Y 568.6,Z 826.441,A -85,B 0,C 180,E1 2443.429,E2 2443.429} C_VEL
LIN {X 0,Y 569.049,Z 805.16,A -85,B 0,C 180,E1 2447.187,E2 2447.187} C_VEL
LIN {X 0,Y 569.733,Z 779.858,A -85,B 0,C 180,E1 2450.546,E2 2450.546} C_VEL
LIN {X 0,Y 570.648,Z 750.117,A -85,B 0,C 180,E1 2453.58,E2 2453.58} C_VEL
LIN {X 0,Y 571.758,Z 716.073,A -85,B 0,C 180,E1 2456.224,E2 2456.224} C_VEL
LIN {X 0,Y 572.795,Z 681.415,A -85,B 0,C 180,E1 2458.223,E2 2458.223} C_VEL
LIN {X 0,Y 573.644,Z 645.331,A -85,B 0,C 180,E1 2459.697,E2 2459.697} C_VEL
LIN {X 0,Y 574.287,Z 607.366,A -85,B 0,C 180,E1 2460.654,E2 2460.654} C_VEL
LIN {X 0,Y 573.652,Z 563.105,A -85,B 0,C 180,E1 2461.352,E2 2461.352} C_VEL
LIN {X 0,Y 567.846,Z 549.53,A -85,B 0,C 180,E1 2461.956,E2 2461.956} C_VEL
LIN {X 0,Y 567.986,Z 549.53,A -85,B 0,C 180,E1 2467.668,E2 2467.668} C_VEL
LIN {X 0,Y 567.748,Z 549.53,A -85,B 0,C 180,E1 2474.137,E2 2474.137} C_VEL
LIN {X 0,Y 567.819,Z 549.53,A -85,B 0,C 180,E1 2478.36,E2 2478.36} C_VEL
LIN {X 0,Y 567.829,Z 549.53,A -85,B 0,C 180,E1 2484.216,E2 2484.216} C_VEL
LIN {X 0,Y 567.813,Z 549.53,A -85,B 0,C 180,E1 2489.666,E2 2489.666} C_VEL
LIN {X 0,Y 567.895,Z 549.53,A -85,B 0,C 180,E1 2494.832,E2 2494.832} C_VEL
LIN {X 0,Y 567.999,Z 549.53,A -85,B 0,C 180,E1 2499.787,E2 2499.787} C_VEL
LIN {X 0,Y 567.899,Z 549.53,A -85,B 0,C 180,E1 2504.581,E2 2504.581} C_VEL
LIN {X 0,Y 567.973,Z 549.53,A -85,B 0,C 180,E1 2510.817,E2 2510.817} C_VEL
LIN {X 0,Y 568.074,Z 549.53,A -85,B 0,C 180,E1 2515.418,E2 2515.418} C_VEL
LIN {X 0,Y 568.147,Z 549.53,A -85,B 0,C 180,E1 2519.987,E2 2519.987} C_VEL
LIN {X 0,Y 568.113,Z 549.53,A -85,B 0,C 180,E1 2524.557,E2 2524.557} C_VEL
LIN {X 0,Y 568.107,Z 549.53,A -85,B 0,C 180,E1 2529.155,E2 2529.155} C_VEL
LIN {X 0,Y 568.132,Z 549.53,A -85,B 0,C 180,E1 2533.814,E2 2533.814} C_VEL
LIN {X 0,Y 568.053,Z 549.53,A -85,B 0,C 180,E1 2538.571,E2 2538.571} C_VEL
LIN {X 0,Y 567.938,Z 549.53,A -85,B 0,C 180,E1 2543.468,E2 2543.468} C_VEL
LIN {X 0,Y 567.844,Z 549.53,A -85,B 0,C 180,E1 2548.72,E2 2548.72} C_VEL
LIN {X 0,Y 568.002,Z 549.53,A -85,B 0,C 180,E1 2554.553,E2 2554.553} C_VEL
LIN {X 0,Y 567.873,Z 549.53,A -85,B 0,C 180,E1 2559.597,E2 2559.597} C_VEL
LIN {X 0,Y 567.67,Z 549.53,A -85,B 0,C 180,E1 2565.835,E2 2565.835} C_VEL
LIN {X 0,Y 567.838,Z 549.53,A -85,B 0,C 180,E1 2570.378,E2 2570.378} C_VEL
LIN {X 0,Y 567.998,Z 549.53,A -85,B 0,C 180,E1 2576.087,E2 2576.087} C_VEL
LIN {X 0,Y 567.855,Z 549.53,A -85,B 0,C 180,E1 2581.422,E2 2581.422} C_VEL
LIN {X 0,Y 567.92,Z 549.53,A -85,B 0,C 180,E1 2586.51,E2 2586.51} C_VEL
LIN {X 0,Y 568.023,Z 549.53,A -85,B 0,C 180,E1 2592.927,E2 2592.927} C_VEL
LIN {X 0,Y 568.047,Z 549.53,A -85,B 0,C 180,E1 2597.729,E2 2597.729} C_VEL
LIN {X 0,Y 568.108,Z 549.53,A -85,B 0,C 180,E1 2602.367,E2 2602.367} C_VEL
LIN {X 0,Y 568.245,Z 549.53,A -85,B 0,C 180,E1 2606.954,E2 2606.954} C_VEL
LIN {X 0,Y 568.047,Z 549.53,A -85,B 0,C 180,E1 2609.076,E2 2609.076} C_VEL
LIN {X 0,Y 572.655,Z 565.362,A -85,B 0,C 180,E1 2609.595,E2 2609.595} C_VEL
LIN {X 0,Y 572.116,Z 602.896,A -85,B 0,C 180,E1 2610.66,E2 2610.66} C_VEL
LIN {X 0,Y 571.311,Z 639.6,A -85,B 0,C 180,E1 2612.364,E2 2612.364} C_VEL
LIN {X 0,Y 570.421,Z 673.371,A -85,B 0,C 180,E1 2614.646,E2 2614.646} C_VEL
LIN {X 0,Y 569.673,Z 702.682,A -85,B 0,C 180,E1 2617.341,E2 2617.341} C_VEL
LIN {X 0,Y 569.071,Z 728.322,A -85,B 0,C 180,E1 2620.503,E2 2620.503} C_VEL
LIN {X 0,Y 568.665,Z 748.114,A -85,B 0,C 180,E1 2623.816,E2 2623.816} C_VEL
LIN {X 0,Y 568.441,Z 763.561,A -85,B 0,C 180,E1 2627.498,E2 2627.498} C_VEL
LIN {X 0,Y 568.336,Z 772.663,A -85,B 0,C 180,E1 2630.955,E2 2630.955} C_VEL
LIN {X 0,Y 568.205,Z 776.306,A -85,B 0,C 180,E1 2633.475,E2 2633.475} C_VEL
LIN {X 0,Y 568.18,Z 777.313,A -85,B 0,C 180,E1 2636.839,E2 2636.839} C_VEL
LIN {X 0,Y 568.369,Z 773.133,A -85,B 0,C 180,E1 2640.723,E2 2640.723} C_VEL
LIN {X 0,Y 568.477,Z 764.044,A -85,B 0,C 180,E1 2644.272,E2 2644.272} C_VEL
LIN {X 0,Y 568.687,Z 748.933,A -85,B 0,C 180,E1 2647.931,E2 2647.931} C_VEL
LIN {X 0,Y 569.023,Z 728.66,A -85,B 0,C 180,E1 2651.359,E2 2651.359} C_VEL
LIN {X 0,Y 569.637,Z 702.292,A -85,B 0,C 180,E1 2654.611,E2 2654.611} C_VEL
LIN {X 0,Y 570.474,Z 673.213,A -85,B 0,C 180,E1 2657.275,E2 2657.275} C_VEL
LIN {X 0,Y 571.379,Z 639.054,A -85,B 0,C 180,E1 2659.573,E2 2659.573} C_VEL
LIN {X 0,Y 572.148,Z 604.063,A -85,B 0,C 180,E1 2661.204,E2 2661.204} C_VEL
LIN {X 0,Y 572.682,Z 567.63,A -85,B 0,C 180,E1 2662.265,E2 2662.265} C_VEL
LIN {X 0,Y 571.365,Z 558.876,A -85,B 0,C 180,E1 2662.502,E2 2662.502} C_VEL
LIN {X 0,Y 568.138,Z 549.53,A -85,B 0,C 180,E1 2662.826,E2 2662.826} C_VEL
LIN {X 0,Y 567.809,Z 549.53,A -85,B 0,C 180,E1 2669.695,E2 2669.695} C_VEL
LIN {X 0,Y 567.871,Z 549.53,A -85,B 0,C 180,E1 2674.859,E2 2674.859} C_VEL
LIN {X 0,Y 568.045,Z 549.53,A -85,B 0,C 180,E1 2679.816,E2 2679.816} C_VEL
LIN {X 0,Y 567.864,Z 549.53,A -85,B 0,C 180,E1 2684.606,E2 2684.606} C_VEL
LIN {X 0,Y 567.979,Z 549.53,A -85,B 0,C 180,E1 2690.842,E2 2690.842} C_VEL
LIN {X 0,Y 568.081,Z 549.53,A -85,B 0,C 180,E1 2695.443,E2 2695.443} C_VEL
LIN {X 0,Y 568.141,Z 549.53,A -85,B 0,C 180,E1 2700.013,E2 2700.013} C_VEL
LIN {X 0,Y 568.115,Z 549.53,A -85,B 0,C 180,E1 2704.582,E2 2704.582} C_VEL
LIN {X 0,Y 568.106,Z 549.53,A -85,B 0,C 180,E1 2709.241,E2 2709.241} C_VEL
LIN {X 0,Y 568.051,Z 549.53,A -85,B 0,C 180,E1 2712.671,E2 2712.671} C_VEL
LIN {X 0,Y 566.761,Z 549.53,A -85,B 0,C 180,E1 2713.542,E2 2713.542} C_VEL
LIN {X 0,Y 560.091,Z 549.53,A -85,B 0,C 180,E1 2715.912,E2 2715.912} C_VEL
LIN {X 0,Y 560.001,Z 549.53,A -85,B 0,C 180,E1 2716.136,E2 2716.136} C_VEL
LIN {X 0,Y 560.014,Z 549.53,A -85,B 0,C 180,E1 2720.514,E2 2720.514} C_VEL
LIN {X 0,Y 559.885,Z 549.53,A -85,B 0,C 180,E1 2725.554,E2 2725.554} C_VEL
LIN {X 0,Y 559.953,Z 549.53,A -85,B 0,C 180,E1 2730.806,E2 2730.806} C_VEL
LIN {X 0,Y 560.055,Z 549.53,A -85,B 0,C 180,E1 2736.36,E2 2736.36} C_VEL
LIN {X 0,Y 559.812,Z 549.53,A -85,B 0,C 180,E1 2742.373,E2 2742.373} C_VEL
LIN {X 0,Y 559.844,Z 549.53,A -85,B 0,C 180,E1 2747.636,E2 2747.636} C_VEL
LIN {X 0,Y 560.072,Z 549.53,A -85,B 0,C 180,E1 2753.933,E2 2753.933} C_VEL
LIN {X 0,Y 560.147,Z 549.53,A -85,B 0,C 180,E1 2757.569,E2 2757.569} C_VEL
LIN {X 0,Y 567.419,Z 567.296,A -85,B 0,C 180,E1 2758.325,E2 2758.325} C_VEL
LIN {X 0,Y 567.195,Z 624.624,A -85,B 0,C 180,E1 2759.3,E2 2759.3} C_VEL
LIN {X 0,Y 566.343,Z 663.312,A -85,B 0,C 180,E1 2760.57,E2 2760.57} C_VEL
LIN {X 0,Y 565.126,Z 700.608,A -85,B 0,C 180,E1 2762.43,E2 2762.43} C_VEL
LIN {X 0,Y 563.734,Z 736.584,A -85,B 0,C 180,E1 2764.93,E2 2764.93} C_VEL
LIN {X 0,Y 562.588,Z 767.115,A -85,B 0,C 180,E1 2767.745,E2 2767.745} C_VEL
LIN {X 0,Y 561.611,Z 794.687,A -85,B 0,C 180,E1 2771.048,E2 2771.048} C_VEL
LIN {X 0,Y 560.927,Z 816.176,A -85,B 0,C 180,E1 2774.395,E2 2774.395} C_VEL
LIN {X 0,Y 560.566,Z 833.447,A -85,B 0,C 180,E1 2777.959,E2 2777.959} C_VEL
LIN {X 0,Y 560.458,Z 846.72,A -85,B 0,C 180,E1 2781.875,E2 2781.875} C_VEL
LIN {X 0,Y 560.335,Z 853.958,A -85,B 0,C 180,E1 2785.367,E2 2785.367} C_VEL
LIN {X 0,Y 560.359,Z 857.088,A -85,B 0,C 180,E1 2788.458,E2 2788.458} C_VEL
LIN {X 0,Y 560.488,Z 857.086,A -85,B 0,C 180,E1 2791.544,E2 2791.544} C_VEL
LIN {X 0,Y 560.452,Z 852.833,A -85,B 0,C 180,E1 2795.359,E2 2795.359} C_VEL
LIN {X 0,Y 560.515,Z 843.299,A -85,B 0,C 180,E1 2799.297,E2 2799.297} C_VEL
LIN {X 0,Y 560.772,Z 828.276,A -85,B 0,C 180,E1 2803.224,E2 2803.224} C_VEL
LIN {X 0,Y 561.221,Z 807.911,A -85,B 0,C 180,E1 2807.003,E2 2807.003} C_VEL
LIN {X 0,Y 562.069,Z 781.603,A -85,B 0,C 180,E1 2810.634,E2 2810.634} C_VEL
LIN {X 0,Y 563.188,Z 750.97,A -85,B 0,C 180,E1 2813.834,E2 2813.834} C_VEL
LIN {X 0,Y 564.404,Z 718.186,A -85,B 0,C 180,E1 2816.443,E2 2816.443} C_VEL
LIN {X 0,Y 565.685,Z 683.203,A -85,B 0,C 180,E1 2818.519,E2 2818.519} C_VEL
LIN {X 0,Y 566.719,Z 646.429,A -85,B 0,C 180,E1 2820.06,E2 2820.06} C_VEL
LIN {X 0,Y 567.487,Z 610.293,A -85,B 0,C 180,E1 2821.011,E2 2821.011} C_VEL
LIN {X 0,Y 567.081,Z 566.11,A -85,B 0,C 180,E1 2821.714,E2 2821.714} C_VEL
LIN {X 0,Y 559.845,Z 549.53,A -85,B 0,C 180,E1 2822.454,E2 2822.454} C_VEL
LIN {X 0,Y 559.973,Z 549.53,A -85,B 0,C 180,E1 2828.303,E2 2828.303} C_VEL
LIN {X 0,Y 559.819,Z 549.53,A -85,B 0,C 180,E1 2834.496,E2 2834.496} C_VEL
LIN {X 0,Y 559.84,Z 549.53,A -85,B 0,C 180,E1 2839.686,E2 2839.686} C_VEL
LIN {X 0,Y 559.806,Z 549.53,A -85,B 0,C 180,E1 2845.517,E2 2845.517} C_VEL
LIN {X 0,Y 559.841,Z 549.53,A -85,B 0,C 180,E1 2850.969,E2 2850.969} C_VEL
LIN {X 0,Y 559.917,Z 549.53,A -85,B 0,C 180,E1 2856.397,E2 2856.397} C_VEL
LIN {X 0,Y 560.12,Z 549.53,A -85,B 0,C 180,E1 2861.129,E2 2861.129} C_VEL
LIN {X 0,Y 559.827,Z 549.53,A -85,B 0,C 180,E1 2866.025,E2 2866.025} C_VEL
LIN {X 0,Y 560.07,Z 549.53,A -85,B 0,C 180,E1 2870.686,E2 2870.686} C_VEL
LIN {X 0,Y 560.187,Z 549.53,A -85,B 0,C 180,E1 2875.353,E2 2875.353} C_VEL
LIN {X 0,Y 560.246,Z 549.53,A -85,B 0,C 180,E1 2879.987,E2 2879.987} C_VEL
LIN {X 0,Y 560.195,Z 549.53,A -85,B 0,C 180,E1 2884.656,E2 2884.656} C_VEL
LIN {X 0,Y 560.21,Z 549.53,A -85,B 0,C 180,E1 2889.286,E2 2889.286} C_VEL
LIN {X 0,Y 560.159,Z 549.53,A -85,B 0,C 180,E1 2894.111,E2 2894.111} C_VEL
LIN {X 0,Y 560.039,Z 549.53,A -85,B 0,C 180,E1 2899.423,E2 2899.423} C_VEL
LIN {X 0,Y 559.993,Z 549.53,A -85,B 0,C 180,E1 2903.821,E2 2903.821} C_VEL
LIN {X 0,Y 559.913,Z 549.53,A -85,B 0,C 180,E1 2908.998,E2 2908.998} C_VEL
LIN {X 0,Y 560.103,Z 549.53,A -85,B 0,C 180,E1 2914.431,E2 2914.431} C_VEL
LIN {X 0,Y 559.878,Z 549.53,A -85,B 0,C 180,E1 2920.277,E2 2920.277} C_VEL
LIN {X 0,Y 559.731,Z 549.53,A -85,B 0,C 180,E1 2925.495,E2 2925.495} C_VEL
LIN {X 0,Y 559.891,Z 549.53,A -85,B 0,C 180,E1 2931.37,E2 2931.37} C_VEL
LIN {X 0,Y 560.065,Z 549.53,A -85,B 0,C 180,E1 2936.598,E2 2936.598} C_VEL
LIN {X 0,Y 559.948,Z 549.53,A -85,B 0,C 180,E1 2940.981,E2 2940.981} C_VEL
LIN {X 0,Y 560.005,Z 549.53,A -85,B 0,C 180,E1 2946.311,E2 2946.311} C_VEL
LIN {X 0,Y 560.124,Z 549.53,A -85,B 0,C 180,E1 2952.76,E2 2952.76} C_VEL
LIN {X 0,Y 560.132,Z 549.53,A -85,B 0,C 180,E1 2957.553,E2 2957.553} C_VEL
LIN {X 0,Y 560.203,Z 549.53,A -85,B 0,C 180,E1 2962.258,E2 2962.258} C_VEL
LIN {X 0,Y 560.337,Z 549.53,A -85,B 0,C 180,E1 2966.911,E2 2966.911} C_VEL
LIN {X 0,Y 560.242,Z 550.339,A -85,B 0,C 180,E1 2968.697,E2 2968.697} C_VEL
LIN {X 0,Y 565.551,Z 567.387,A -85,B 0,C 180,E1 2969.282,E2 2969.282} C_VEL
LIN {X 0,Y 564.87,Z 604.711,A -85,B 0,C 180,E1 2970.382,E2 2970.382} C_VEL
LIN {X 0,Y 563.948,Z 640.759,A -85,B 0,C 180,E1 2972.107,E2 2972.107} C_VEL
LIN {X 0,Y 562.885,Z 674.26,A -85,B 0,C 180,E1 2974.419,E2 2974.419} C_VEL
LIN {X 0,Y 561.989,Z 704.454,A -85,B 0,C 180,E1 2977.266,E2 2977.266} C_VEL
LIN {X 0,Y 561.278,Z 729.467,A -85,B 0,C 180,E1 2980.455,E2 2980.455} C_VEL
LIN {X 0,Y 560.837,Z 747.976,A -85,B 0,C 180,E1 2983.616,E2 2983.616} C_VEL
LIN {X 0,Y 560.614,Z 763.022,A -85,B 0,C 180,E1 2987.222,E2 2987.222} C_VEL
LIN {X 0,Y 560.462,Z 771.87,A -85,B 0,C 180,E1 2990.487,E2 2990.487} C_VEL
LIN {X 0,Y 560.274,Z 776.629,A -85,B 0,C 180,E1 2993.827,E2 2993.827} C_VEL
LIN {X 0,Y 560.273,Z 777.121,A -85,B 0,C 180,E1 2997.331,E2 2997.331} C_VEL
LIN {X 0,Y 560.471,Z 773.182,A -85,B 0,C 180,E1 3000.766,E2 3000.766} C_VEL
LIN {X 0,Y 560.588,Z 763.939,A -85,B 0,C 180,E1 3004.421,E2 3004.421} C_VEL
LIN {X 0,Y 560.832,Z 748.29,A -85,B 0,C 180,E1 3008.231,E2 3008.231} C_VEL
LIN {X 0,Y 561.284,Z 728.033,A -85,B 0,C 180,E1 3011.671,E2 3011.671} C_VEL
LIN {X 0,Y 561.994,Z 702.608,A -85,B 0,C 180,E1 3014.841,E2 3014.841} C_VEL
LIN {X 0,Y 562.962,Z 672.846,A -85,B 0,C 180,E1 3017.603,E2 3017.603} C_VEL
LIN {X 0,Y 564.052,Z 639.202,A -85,B 0,C 180,E1 3019.891,E2 3019.891} C_VEL
LIN {X 0,Y 564.976,Z 603.288,A -85,B 0,C 180,E1 3021.577,E2 3021.577} C_VEL
LIN {X 0,Y 565.593,Z 567.191,A -85,B 0,C 180,E1 3022.63,E2 3022.63} C_VEL
LIN {X 0,Y 563.129,Z 557.972,A -85,B 0,C 180,E1 3022.936,E2 3022.936} C_VEL
LIN {X 0,Y 560.144,Z 549.53,A -85,B 0,C 180,E1 3023.326,E2 3023.326} C_VEL
LIN {X 0,Y 559.901,Z 549.53,A -85,B 0,C 180,E1 3029.59,E2 3029.59} C_VEL
LIN {X 0,Y 559.95,Z 549.53,A -85,B 0,C 180,E1 3034.478,E2 3034.478} C_VEL
LIN {X 0,Y 560.122,Z 549.53,A -85,B 0,C 180,E1 3040.546,E2 3040.546} C_VEL
LIN {X 0,Y 559.97,Z 549.53,A -85,B 0,C 180,E1 3044.384,E2 3044.384} C_VEL
LIN {X 0,Y 560.073,Z 549.53,A -85,B 0,C 180,E1 3050.712,E2 3050.712} C_VEL
LIN {X 0,Y 560.195,Z 549.53,A -85,B 0,C 180,E1 3055.379,E2 3055.379} C_VEL
LIN {X 0,Y 560.239,Z 549.53,A -85,B 0,C 180,E1 3060.013,E2 3060.013} C_VEL
LIN {X 0,Y 560.195,Z 549.53,A -85,B 0,C 180,E1 3064.685,E2 3064.685} C_VEL
LIN {X 0,Y 560.203,Z 549.53,A -85,B 0,C 180,E1 3069.312,E2 3069.312} C_VEL
LIN {X 0,Y 560.181,Z 549.53,A -85,B 0,C 180,E1 3074.13,E2 3074.13} C_VEL
LIN {X 0,Y 560.001,Z 549.53,A -85,B 0,C 180,E1 3076.136,E2 3076.136} C_VEL
LIN {X 0,Y 557.542,Z 549.53,A -85,B 0,C 180,E1 3077.453,E2 3077.453} C_VEL
LIN {X 0,Y 552.106,Z 549.53,A -85,B 0,C 180,E1 3079.652,E2 3079.652} C_VEL
LIN {X 0,Y 551.991,Z 549.53,A -85,B 0,C 180,E1 3085.562,E2 3085.562} C_VEL
LIN {X 0,Y 552.023,Z 549.53,A -85,B 0,C 180,E1 3091.298,E2 3091.298} C_VEL
LIN {X 0,Y 552.042,Z 549.53,A -85,B 0,C 180,E1 3096.974,E2 3096.974} C_VEL
LIN {X 0,Y 551.848,Z 549.53,A -85,B 0,C 180,E1 3103.132,E2 3103.132} C_VEL
LIN {X 0,Y 551.971,Z 549.53,A -85,B 0,C 180,E1 3108.996,E2 3108.996} C_VEL
LIN {X 0,Y 552.167,Z 549.53,A -85,B 0,C 180,E1 3115.075,E2 3115.075} C_VEL
LIN {X 0,Y 552.217,Z 549.804,A -85,B 0,C 180,E1 3117.081,E2 3117.081} C_VEL
LIN {X 0,Y 560.699,Z 569.433,A -85,B 0,C 180,E1 3117.932,E2 3117.932} C_VEL
LIN {X 0,Y 560.37,Z 625.233,A -85,B 0,C 180,E1 3118.902,E2 3118.902} C_VEL
LIN {X 0,Y 559.364,Z 663.664,A -85,B 0,C 180,E1 3120.182,E2 3120.182} C_VEL
LIN {X 0,Y 557.951,Z 701.34,A -85,B 0,C 180,E1 3122.092,E2 3122.092} C_VEL
LIN {X 0,Y 556.432,Z 736.011,A -85,B 0,C 180,E1 3124.529,E2 3124.529} C_VEL
LIN {X 0,Y 555.051,Z 767.244,A -85,B 0,C 180,E1 3127.44,E2 3127.44} C_VEL
LIN {X 0,Y 553.931,Z 793.931,A -85,B 0,C 180,E1 3130.669,E2 3130.669} C_VEL
LIN {X 0,Y 553.099,Z 816.177,A -85,B 0,C 180,E1 3134.169,E2 3134.169} C_VEL
LIN {X 0,Y 552.732,Z 833.448,A -85,B 0,C 180,E1 3137.786,E2 3137.786} C_VEL
LIN {X 0,Y 552.594,Z 846.72,A -85,B 0,C 180,E1 3141.759,E2 3141.759} C_VEL
LIN {X 0,Y 552.457,Z 853.958,A -85,B 0,C 180,E1 3145.301,E2 3145.301} C_VEL
LIN {X 0,Y 552.463,Z 857.088,A -85,B 0,C 180,E1 3148.436,E2 3148.436} C_VEL
LIN {X 0,Y 552.583,Z 857.086,A -85,B 0,C 180,E1 3151.566,E2 3151.566} C_VEL
LIN {X 0,Y 552.544,Z 852.754,A -85,B 0,C 180,E1 3155.486,E2 3155.486} C_VEL
LIN {X 0,Y 552.616,Z 843.299,A -85,B 0,C 180,E1 3159.431,E2 3159.431} C_VEL
LIN {X 0,Y 552.922,Z 828.276,A -85,B 0,C 180,E1 3163.415,E2 3163.415} C_VEL
LIN {X 0,Y 553.488,Z 806.988,A -85,B 0,C 180,E1 3167.402,E2 3167.402} C_VEL
LIN {X 0,Y 554.456,Z 781.602,A -85,B 0,C 180,E1 3170.93,E2 3170.93} C_VEL
LIN {X 0,Y 555.809,Z 750.971,A -85,B 0,C 180,E1 3174.17,E2 3174.17} C_VEL
LIN {X 0,Y 557.194,Z 717.814,A -85,B 0,C 180,E1 3176.839,E2 3176.839} C_VEL
LIN {X 0,Y 558.632,Z 683.7,A -85,B 0,C 180,E1 3178.887,E2 3178.887} C_VEL
LIN {X 0,Y 559.836,Z 646.385,A -85,B 0,C 180,E1 3180.47,E2 3180.47} C_VEL
LIN {X 0,Y 560.714,Z 609.418,A -85,B 0,C 180,E1 3181.444,E2 3181.444} C_VEL
LIN {X 0,Y 560.111,Z 568.068,A -85,B 0,C 180,E1 3182.126,E2 3182.126} C_VEL
LIN {X 0,Y 551.922,Z 549.53,A -85,B 0,C 180,E1 3183.008,E2 3183.008} C_VEL
LIN {X 0,Y 552.001,Z 549.53,A -85,B 0,C 180,E1 3188.96,E2 3188.96} C_VEL
LIN {X 0,Y 551.944,Z 549.53,A -85,B 0,C 180,E1 3195.305,E2 3195.305} C_VEL
LIN {X 0,Y 551.959,Z 549.53,A -85,B 0,C 180,E1 3201.032,E2 3201.032} C_VEL
LIN {X 0,Y 551.855,Z 549.53,A -85,B 0,C 180,E1 3206.84,E2 3206.84} C_VEL
LIN {X 0,Y 551.91,Z 549.53,A -85,B 0,C 180,E1 3212.295,E2 3212.295} C_VEL
LIN {X 0,Y 552.036,Z 549.53,A -85,B 0,C 180,E1 3218.345,E2 3218.345} C_VEL
LIN {X 0,Y 552.234,Z 549.53,A -85,B 0,C 180,E1 3223.022,E2 3223.022} C_VEL
LIN {X 0,Y 552.162,Z 549.53,A -85,B 0,C 180,E1 3229.695,E2 3229.695} C_VEL
LIN {X 0,Y 552.289,Z 549.53,A -85,B 0,C 180,E1 3235.286,E2 3235.286} C_VEL
LIN {X 0,Y 552.348,Z 549.53,A -85,B 0,C 180,E1 3239.987,E2 3239.987} C_VEL
LIN {X 0,Y 552.317,Z 549.53,A -85,B 0,C 180,E1 3244.687,E2 3244.687} C_VEL
LIN {X 0,Y 552.17,Z 549.53,A -85,B 0,C 180,E1 3250.309,E2 3250.309} C_VEL
LIN {X 0,Y 552.114,Z 549.53,A -85,B 0,C 180,E1 3255.844,E2 3255.844} C_VEL
LIN {X 0,Y 552.073,Z 549.53,A -85,B 0,C 180,E1 3261.665,E2 3261.665} C_VEL
LIN {X 0,Y 551.978,Z 549.53,A -85,B 0,C 180,E1 3267.672,E2 3267.672} C_VEL
LIN {X 0,Y 552.156,Z 549.53,A -85,B 0,C 180,E1 3273.109,E2 3273.109} C_VEL
LIN {X 0,Y 551.993,Z 549.53,A -85,B 0,C 180,E1 3278.931,E2 3278.931} C_VEL
LIN {X 0,Y 551.823,Z 549.53,A -85,B 0,C 180,E1 3284.682,E2 3284.682} C_VEL
LIN {X 0,Y 551.942,Z 549.53,A -85,B 0,C 180,E1 3289.917,E2 3289.917} C_VEL
LIN {X 0,Y 552.192,Z 549.53,A -85,B 0,C 180,E1 3295.026,E2 3295.026} C_VEL
LIN {X 0,Y 552.071,Z 549.53,A -85,B 0,C 180,E1 3300.956,E2 3300.956} C_VEL
LIN {X 0,Y 552.006,Z 549.53,A -85,B 0,C 180,E1 3305.791,E2 3305.791} C_VEL
LIN {X 0,Y 552.118,Z 549.53,A -85,B 0,C 180,E1 3310.853,E2 3310.853} C_VEL
LIN {X 0,Y 552.246,Z 549.53,A -85,B 0,C 180,E1 3315.762,E2 3315.762} C_VEL
LIN {X 0,Y 552.288,Z 549.53,A -85,B 0,C 180,E1 3322.147,E2 3322.147} C_VEL
LIN {X 0,Y 552.326,Z 549.53,A -85,B 0,C 180,E1 3328.042,E2 3328.042} C_VEL
LIN {X 0,Y 552.325,Z 549.53,A -85,B 0,C 180,E1 3328.237,E2 3328.237} C_VEL
LIN {X 0,Y 558.447,Z 569.472,A -85,B 0,C 180,E1 3328.962,E2 3328.962} C_VEL
LIN {X 0,Y 557.651,Z 607.703,A -85,B 0,C 180,E1 3330.144,E2 3330.144} C_VEL
LIN {X 0,Y 556.51,Z 643.523,A -85,B 0,C 180,E1 3331.941,E2 3331.941} C_VEL
LIN {X 0,Y 555.325,Z 676.326,A -85,B 0,C 180,E1 3334.284,E2 3334.284} C_VEL
LIN {X 0,Y 554.307,Z 705.642,A -85,B 0,C 180,E1 3337.135,E2 3337.135} C_VEL
LIN {X 0,Y 553.481,Z 730.612,A -85,B 0,C 180,E1 3340.405,E2 3340.405} C_VEL
LIN {X 0,Y 552.968,Z 749.809,A -85,B 0,C 180,E1 3343.813,E2 3343.813} C_VEL
LIN {X 0,Y 552.673,Z 764.31,A -85,B 0,C 180,E1 3347.477,E2 3347.477} C_VEL
LIN {X 0,Y 552.532,Z 772.63,A -85,B 0,C 180,E1 3350.795,E2 3350.795} C_VEL
LIN {X 0,Y 552.334,Z 776.886,A -85,B 0,C 180,E1 3354.192,E2 3354.192} C_VEL
LIN {X 0,Y 552.373,Z 776.916,A -85,B 0,C 180,E1 3357.671,E2 3357.671} C_VEL
LIN {X 0,Y 552.551,Z 772.353,A -85,B 0,C 180,E1 3361.256,E2 3361.256} C_VEL
LIN {X 0,Y 552.683,Z 762.241,A -85,B 0,C 180,E1 3365.047,E2 3365.047} C_VEL
LIN {X 0,Y 552.994,Z 746.015,A -85,B 0,C 180,E1 3368.874,E2 3368.874} C_VEL
LIN {X 0,Y 553.577,Z 724.093,A -85,B 0,C 180,E1 3372.46,E2 3372.46} C_VEL
LIN {X 0,Y 554.529,Z 698.206,A -85,B 0,C 180,E1 3375.581,E2 3375.581} C_VEL
LIN {X 0,Y 555.686,Z 667.329,A -85,B 0,C 180,E1 3378.345,E2 3378.345} C_VEL
LIN {X 0,Y 556.894,Z 634.669,A -85,B 0,C 180,E1 3380.475,E2 3380.475} C_VEL
LIN {X 0,Y 557.941,Z 599.921,A -85,B 0,C 180,E1 3382.055,E2 3382.055} C_VEL
LIN {X 0,Y 557.977,Z 565.076,A -85,B 0,C 180,E1 3383.07,E2 3383.07} C_VEL
LIN {X 0,Y 552.183,Z 549.53,A -85,B 0,C 180,E1 3383.698,E2 3383.698} C_VEL
LIN {X 0,Y 551.891,Z 549.53,A -85,B 0,C 180,E1 3388.724,E2 3388.724} C_VEL
LIN {X 0,Y 552.047,Z 549.53,A -85,B 0,C 180,E1 3394.426,E2 3394.426} C_VEL
LIN {X 0,Y 552.245,Z 549.53,A -85,B 0,C 180,E1 3400.877,E2 3400.877} C_VEL
LIN {X 0,Y 551.918,Z 549.53,A -85,B 0,C 180,E1 3405.772,E2 3405.772} C_VEL
LIN {X 0,Y 552.159,Z 549.53,A -85,B 0,C 180,E1 3410.578,E2 3410.578} C_VEL
LIN {X 0,Y 552.332,Z 549.53,A -85,B 0,C 180,E1 3415.313,E2 3415.313} C_VEL
LIN {X 0,Y 552.341,Z 549.53,A -85,B 0,C 180,E1 3420.013,E2 3420.013} C_VEL
LIN {X 0,Y 552.318,Z 549.53,A -85,B 0,C 180,E1 3424.713,E2 3424.713} C_VEL
LIN {X 0,Y 552.168,Z 549.53,A -85,B 0,C 180,E1 3430.321,E2 3430.321} C_VEL
LIN {X 0,Y 552.105,Z 549.53,A -85,B 0,C 180,E1 3436.139,E2 3436.139} C_VEL
LIN {X 0,Y 552.106,Z 549.53,A -85,B 0,C 180,E1 3439.652,E2 3439.652} C_VEL
LIN {X 0,Y 548.079,Z 549.53,A -85,B 0,C 180,E1 3441.421,E2 3441.421} C_VEL
LIN {X 0,Y 544.099,Z 549.53,A -85,B 0,C 180,E1 3443.215,E2 3443.215} C_VEL
LIN {X 0,Y 544.085,Z 549.53,A -85,B 0,C 180,E1 3448.139,E2 3448.139} C_VEL
LIN {X 0,Y 544.211,Z 549.53,A -85,B 0,C 180,E1 3453.713,E2 3453.713} C_VEL
LIN {X 0,Y 544.009,Z 549.53,A -85,B 0,C 180,E1 3459.648,E2 3459.648} C_VEL
LIN {X 0,Y 543.945,Z 549.53,A -85,B 0,C 180,E1 3466.166,E2 3466.166} C_VEL
LIN {X 0,Y 544.133,Z 549.53,A -85,B 0,C 180,E1 3472.404,E2 3472.404} C_VEL
LIN {X 0,Y 544.29,Z 549.53,A -85,B 0,C 180,E1 3476.512,E2 3476.512} C_VEL
LIN {X 0,Y 554.001,Z 572.661,A -85,B 0,C 180,E1 3477.545,E2 3477.545} C_VEL
LIN {X 0,Y 553.604,Z 624.635,A -85,B 0,C 180,E1 3478.461,E2 3478.461} C_VEL
LIN {X 0,Y 552.479,Z 663.156,A -85,B 0,C 180,E1 3479.748,E2 3479.748} C_VEL
LIN {X 0,Y 550.911,Z 700.198,A -85,B 0,C 180,E1 3481.629,E2 3481.629} C_VEL
LIN {X 0,Y 549.106,Z 736.447,A -85,B 0,C 180,E1 3484.203,E2 3484.203} C_VEL
LIN {X 0,Y 547.533,Z 767.049,A -85,B 0,C 180,E1 3487.091,E2 3487.091} C_VEL
LIN {X 0,Y 546.239,Z 794.349,A -85,B 0,C 180,E1 3490.445,E2 3490.445} C_VEL
LIN {X 0,Y 545.297,Z 817.271,A -85,B 0,C 180,E1 3494.142,E2 3494.142} C_VEL
LIN {X 0,Y 544.836,Z 834.986,A -85,B 0,C 180,E1 3498.012,E2 3498.012} C_VEL
LIN {X 0,Y 544.717,Z 846.72,A -85,B 0,C 180,E1 3501.638,E2 3501.638} C_VEL
LIN {X 0,Y 544.557,Z 853.958,A -85,B 0,C 180,E1 3505.233,E2 3505.233} C_VEL
LIN {X 0,Y 544.561,Z 857.088,A -85,B 0,C 180,E1 3508.413,E2 3508.413} C_VEL
LIN {X 0,Y 544.677,Z 857.087,A -85,B 0,C 180,E1 3511.589,E2 3511.589} C_VEL
LIN {X 0,Y 544.652,Z 852.754,A -85,B 0,C 180,E1 3515.566,E2 3515.566} C_VEL
LIN {X 0,Y 544.718,Z 843.3,A -85,B 0,C 180,E1 3519.569,E2 3519.569} C_VEL
LIN {X 0,Y 545.069,Z 828.469,A -85,B 0,C 180,E1 3523.567,E2 3523.567} C_VEL
LIN {X 0,Y 545.725,Z 807.811,A -85,B 0,C 180,E1 3527.519,E2 3527.519} C_VEL
LIN {X 0,Y 546.852,Z 781.734,A -85,B 0,C 180,E1 3531.219,E2 3531.219} C_VEL
LIN {X 0,Y 548.363,Z 751.28,A -85,B 0,C 180,E1 3534.491,E2 3534.491} C_VEL
LIN {X 0,Y 549.971,Z 718.078,A -85,B 0,C 180,E1 3537.202,E2 3537.202} C_VEL
LIN {X 0,Y 551.657,Z 682.142,A -85,B 0,C 180,E1 3539.37,E2 3539.37} C_VEL
LIN {X 0,Y 553.028,Z 645.721,A -85,B 0,C 180,E1 3540.909,E2 3540.909} C_VEL
LIN {X 0,Y 553.967,Z 609.367,A -85,B 0,C 180,E1 3541.873,E2 3541.873} C_VEL
LIN {X 0,Y 553.494,Z 570.824,A -85,B 0,C 180,E1 3542.516,E2 3542.516} C_VEL
LIN {X 0,Y 543.968,Z 549.53,A -85,B 0,C 180,E1 3543.544,E2 3543.544} C_VEL
LIN {X 0,Y 544.089,Z 549.53,A -85,B 0,C 180,E1 3549.048,E2 3549.048} C_VEL
LIN {X 0,Y 543.967,Z 549.53,A -85,B 0,C 180,E1 3553.911,E2 3553.911} C_VEL
LIN {X 0,Y 544.054,Z 549.53,A -85,B 0,C 180,E1 3558.496,E2 3558.496} C_VEL
LIN {X 0,Y 543.976,Z 549.53,A -85,B 0,C 180,E1 3564.363,E2 3564.363} C_VEL
LIN {X 0,Y 543.982,Z 549.53,A -85,B 0,C 180,E1 3570.037,E2 3570.037} C_VEL
LIN {X 0,Y 544.043,Z 549.53,A -85,B 0,C 180,E1 3576.254,E2 3576.254} C_VEL
LIN {X 0,Y 544.317,Z 549.53,A -85,B 0,C 180,E1 3582.235,E2 3582.235} C_VEL
LIN {X 0,Y 544.243,Z 549.53,A -85,B 0,C 180,E1 3588.798,E2 3588.798} C_VEL
LIN {X 0,Y 544.534,Z 549.53,A -85,B 0,C 180,E1 3593.624,E2 3593.624} C_VEL
LIN {X 0,Y 544.447,Z 549.53,A -85,B 0,C 180,E1 3599.987,E2 3599.987} C_VEL
LIN {X 0,Y 544.423,Z 549.53,A -85,B 0,C 180,E1 3604.755,E2 3604.755} C_VEL
LIN {X 0,Y 544.371,Z 549.53,A -85,B 0,C 180,E1 3609.558,E2 3609.558} C_VEL
LIN {X 0,Y 544.336,Z 549.53,A -85,B 0,C 180,E1 3614.431,E2 3614.431} C_VEL
LIN {X 0,Y 544.22,Z 549.53,A -85,B 0,C 180,E1 3619.478,E2 3619.478} C_VEL
LIN {X 0,Y 544.085,Z 549.53,A -85,B 0,C 180,E1 3624.563,E2 3624.563} C_VEL
LIN {X 0,Y 544.061,Z 549.53,A -85,B 0,C 180,E1 3630.701,E2 3630.701} C_VEL
LIN {X 0,Y 544.151,Z 549.53,A -85,B 0,C 180,E1 3635.591,E2 3635.591} C_VEL
LIN {X 0,Y 544.044,Z 549.53,A -85,B 0,C 180,E1 3641.705,E2 3641.705} C_VEL
LIN {X 0,Y 544.04,Z 549.53,A -85,B 0,C 180,E1 3648.46,E2 3648.46} C_VEL
LIN {X 0,Y 544.177,Z 549.53,A -85,B 0,C 180,E1 3654.384,E2 3654.384} C_VEL
LIN {X 0,Y 544.087,Z 549.53,A -85,B 0,C 180,E1 3660.05,E2 3660.05} C_VEL
LIN {X 0,Y 544.072,Z 549.53,A -85,B 0,C 180,E1 3666.181,E2 3666.181} C_VEL
LIN {X 0,Y 544.253,Z 549.53,A -85,B 0,C 180,E1 3672.241,E2 3672.241} C_VEL
LIN {X 0,Y 544.295,Z 549.53,A -85,B 0,C 180,E1 3677.184,E2 3677.184} C_VEL
LIN {X 0,Y 544.372,Z 549.53,A -85,B 0,C 180,E1 3682.032,E2 3682.032} C_VEL
LIN {X 0,Y 544.45,Z 549.53,A -85,B 0,C 180,E1 3687.815,E2 3687.815} C_VEL
LIN {X 0,Y 551.411,Z 569.71,A -85,B 0,C 180,E1 3688.594,E2 3688.594} C_VEL
LIN {X 0,Y 550.488,Z 607.827,A -85,B 0,C 180,E1 3689.789,E2 3689.789} C_VEL
LIN {X 0,Y 549.227,Z 643.061,A -85,B 0,C 180,E1 3691.573,E2 3691.573} C_VEL
LIN {X 0,Y 547.88,Z 676.006,A -85,B 0,C 180,E1 3693.947,E2 3693.947} C_VEL
LIN {X 0,Y 546.61,Z 705.999,A -85,B 0,C 180,E1 3696.903,E2 3696.903} C_VEL
LIN {X 0,Y 545.751,Z 730.207,A -85,B 0,C 180,E1 3700.116,E2 3700.116} C_VEL
LIN {X 0,Y 545.132,Z 749.554,A -85,B 0,C 180,E1 3703.583,E2 3703.583} C_VEL
LIN {X 0,Y 544.8,Z 764.451,A -85,B 0,C 180,E1 3707.396,E2 3707.396} C_VEL
LIN {X 0,Y 544.601,Z 773.376,A -85,B 0,C 180,E1 3711.112,E2 3711.112} C_VEL
LIN {X 0,Y 544.412,Z 777.14,A -85,B 0,C 180,E1 3714.567,E2 3714.567} C_VEL
LIN {X 0,Y 544.476,Z 776.651,A -85,B 0,C 180,E1 3718.108,E2 3718.108} C_VEL
LIN {X 0,Y 544.615,Z 771.514,A -85,B 0,C 180,E1 3721.765,E2 3721.765} C_VEL
LIN {X 0,Y 544.807,Z 760.959,A -85,B 0,C 180,E1 3725.566,E2 3725.566} C_VEL
LIN {X 0,Y 545.175,Z 745.136,A -85,B 0,C 180,E1 3729.23,E2 3729.23} C_VEL
LIN {X 0,Y 545.863,Z 723.851,A -85,B 0,C 180,E1 3732.734,E2 3732.734} C_VEL
LIN {X 0,Y 546.9,Z 698.458,A -85,B 0,C 180,E1 3735.838,E2 3735.838} C_VEL
LIN {X 0,Y 548.279,Z 667.029,A -85,B 0,C 180,E1 3738.688,E2 3738.688} C_VEL
LIN {X 0,Y 549.604,Z 635.08,A -85,B 0,C 180,E1 3740.799,E2 3740.799} C_VEL
LIN {X 0,Y 550.779,Z 601.194,A -85,B 0,C 180,E1 3742.37,E2 3742.37} C_VEL
LIN {X 0,Y 551.005,Z 567.602,A -85,B 0,C 180,E1 3743.385,E2 3743.385} C_VEL
LIN {X 0,Y 544.207,Z 549.53,A -85,B 0,C 180,E1 3744.196,E2 3744.196} C_VEL
LIN {X 0,Y 543.958,Z 549.53,A -85,B 0,C 180,E1 3750.066,E2 3750.066} C_VEL
LIN {X 0,Y 544.055,Z 549.53,A -85,B 0,C 180,E1 3755.436,E2 3755.436} C_VEL
LIN {X 0,Y 544.296,Z 549.53,A -85,B 0,C 180,E1 3760.587,E2 3760.587} C_VEL
LIN {X 0,Y 544.002,Z 549.53,A -85,B 0,C 180,E1 3766.131,E2 3766.131} C_VEL
LIN {X 0,Y 544.275,Z 549.53,A -85,B 0,C 180,E1 3770.44,E2 3770.44} C_VEL
LIN {X 0,Y 544.436,Z 549.53,A -85,B 0,C 180,E1 3775.245,E2 3775.245} C_VEL
LIN {X 0,Y 544.439,Z 549.53,A -85,B 0,C 180,E1 3780.013,E2 3780.013} C_VEL
LIN {X 0,Y 544.423,Z 549.53,A -85,B 0,C 180,E1 3784.782,E2 3784.782} C_VEL
LIN {X 0,Y 544.367,Z 549.53,A -85,B 0,C 180,E1 3789.585,E2 3789.585} C_VEL
LIN {X 0,Y 544.356,Z 549.53,A -85,B 0,C 180,E1 3794.457,E2 3794.457} C_VEL
LIN {X 0,Y 544.204,Z 549.53,A -85,B 0,C 180,E1 3799.64,E2 3799.64} C_VEL
LIN {X 0,Y 544.099,Z 549.53,A -85,B 0,C 180,E1 3803.215,E2 3803.215} C_VEL
LIN {X 0,Y 540.15,Z 549.53,A -85,B 0,C 180,E1 3805.017,E2 3805.017} C_VEL
LIN {X 0,Y 536.112,Z 549.53,A -85,B 0,C 180,E1 3806.845,E2 3806.845} C_VEL
LIN {X 0,Y 536.242,Z 549.53,A -85,B 0,C 180,E1 3812.414,E2 3812.414} C_VEL
LIN {X 0,Y 536.163,Z 549.53,A -85,B 0,C 180,E1 3818.263,E2 3818.263} C_VEL
LIN {X 0,Y 535.917,Z 549.53,A -85,B 0,C 180,E1 3824.749,E2 3824.749} C_VEL
LIN {X 0,Y 536.061,Z 549.53,A -85,B 0,C 180,E1 3829.652,E2 3829.652} C_VEL
LIN {X 0,Y 536.331,Z 549.53,A -85,B 0,C 180,E1 3835.953,E2 3835.953} C_VEL
LIN {X 0,Y 547.329,Z 574.722,A -85,B 0,C 180,E1 3837.132,E2 3837.132} C_VEL
LIN {X 0,Y 546.837,Z 625.793,A -85,B 0,C 180,E1 3838.059,E2 3838.059} C_VEL
LIN {X 0,Y 545.579,Z 663.031,A -85,B 0,C 180,E1 3839.319,E2 3839.319} C_VEL
LIN {X 0,Y 543.853,Z 699.883,A -85,B 0,C 180,E1 3841.205,E2 3841.205} C_VEL
LIN {X 0,Y 541.812,Z 735.67,A -85,B 0,C 180,E1 3843.761,E2 3843.761} C_VEL
LIN {X 0,Y 540.061,Z 767.048,A -85,B 0,C 180,E1 3846.756,E2 3846.756} C_VEL
LIN {X 0,Y 538.593,Z 794.35,A -85,B 0,C 180,E1 3850.156,E2 3850.156} C_VEL
LIN {X 0,Y 537.484,Z 817.272,A -85,B 0,C 180,E1 3853.905,E2 3853.905} C_VEL
LIN {X 0,Y 537.044,Z 833.449,A -85,B 0,C 180,E1 3857.424,E2 3857.424} C_VEL
LIN {X 0,Y 536.818,Z 846.72,A -85,B 0,C 180,E1 3861.515,E2 3861.515} C_VEL
LIN {X 0,Y 536.659,Z 853.959,A -85,B 0,C 180,E1 3865.162,E2 3865.162} C_VEL
LIN {X 0,Y 536.67,Z 857.088,A -85,B 0,C 180,E1 3868.39,E2 3868.39} C_VEL
LIN {X 0,Y 536.801,Z 857.087,A -85,B 0,C 180,E1 3871.612,E2 3871.612} C_VEL
LIN {X 0,Y 536.757,Z 852.754,A -85,B 0,C 180,E1 3875.648,E2 3875.648} C_VEL
LIN {X 0,Y 536.828,Z 843.3,A -85,B 0,C 180,E1 3879.711,E2 3879.711} C_VEL
LIN {X 0,Y 537.256,Z 827.776,A -85,B 0,C 180,E1 3883.933,E2 3883.933} C_VEL
LIN {X 0,Y 538.06,Z 806.657,A -85,B 0,C 180,E1 3887.97,E2 3887.97} C_VEL
LIN {X 0,Y 539.341,Z 780.544,A -85,B 0,C 180,E1 3891.676,E2 3891.676} C_VEL
LIN {X 0,Y 540.989,Z 750.336,A -85,B 0,C 180,E1 3894.938,E2 3894.938} C_VEL
LIN {X 0,Y 542.868,Z 716.592,A -85,B 0,C 180,E1 3897.697,E2 3897.697} C_VEL
LIN {X 0,Y 544.728,Z 680.815,A -85,B 0,C 180,E1 3899.852,E2 3899.852} C_VEL
LIN {X 0,Y 546.259,Z 643.804,A -85,B 0,C 180,E1 3901.403,E2 3901.403} C_VEL
LIN {X 0,Y 547.295,Z 607.548,A -85,B 0,C 180,E1 3902.341,E2 3902.341} C_VEL
LIN {X 0,Y 546.787,Z 573.345,A -85,B 0,C 180,E1 3902.926,E2 3902.926} C_VEL
LIN {X 0,Y 536.041,Z 549.53,A -85,B 0,C 180,E1 3904.093,E2 3904.093} C_VEL
LIN {X 0,Y 536.185,Z 549.53,A -85,B 0,C 180,E1 3908.256,E2 3908.256} C_VEL
LIN {X 0,Y 536.003,Z 549.53,A -85,B 0,C 180,E1 3914.736,E2 3914.736} C_VEL
LIN {X 0,Y 536.067,Z 549.53,A -85,B 0,C 180,E1 3919.645,E2 3919.645} C_VEL
LIN {X 0,Y 536.025,Z 549.53,A -85,B 0,C 180,E1 3924.729,E2 3924.729} C_VEL
LIN {X 0,Y 536.023,Z 549.53,A -85,B 0,C 180,E1 3930.778,E2 3930.778} C_VEL
LIN {X 0,Y 536.142,Z 549.53,A -85,B 0,C 180,E1 3936.785,E2 3936.785} C_VEL
LIN {X 0,Y 536.382,Z 549.53,A -85,B 0,C 180,E1 3941.963,E2 3941.963} C_VEL
LIN {X 0,Y 536.33,Z 549.53,A -85,B 0,C 180,E1 3948.63,E2 3948.63} C_VEL
LIN {X 0,Y 536.602,Z 549.53,A -85,B 0,C 180,E1 3953.529,E2 3953.529} C_VEL
LIN {X 0,Y 536.731,Z 549.53,A -85,B 0,C 180,E1 3958.376,E2 3958.376} C_VEL
LIN {X 0,Y 536.51,Z 549.53,A -85,B 0,C 180,E1 3964.826,E2 3964.826} C_VEL
LIN {X 0,Y 536.391,Z 549.53,A -85,B 0,C 180,E1 3970.047,E2 3970.047} C_VEL
LIN {X 0,Y 536.396,Z 549.53,A -85,B 0,C 180,E1 3974.649,E2 3974.649} C_VEL
LIN {X 0,Y 536.31,Z 549.53,A -85,B 0,C 180,E1 3979.714,E2 3979.714} C_VEL
LIN {X 0,Y 536.078,Z 549.53,A -85,B 0,C 180,E1 3985.738,E2 3985.738} C_VEL
LIN {X 0,Y 536.174,Z 549.53,A -85,B 0,C 180,E1 3990.414,E2 3990.414} C_VEL
LIN {X 0,Y 536.223,Z 549.53,A -85,B 0,C 180,E1 3996.199,E2 3996.199} C_VEL
LIN {X 0,Y 536.017,Z 549.53,A -85,B 0,C 180,E1 4002.475,E2 4002.475} C_VEL
LIN {X 0,Y 536.012,Z 549.53,A -85,B 0,C 180,E1 4007.493,E2 4007.493} C_VEL
LIN {X 0,Y 536.229,Z 549.53,A -85,B 0,C 180,E1 4013.773,E2 4013.773} C_VEL
LIN {X 0,Y 536.195,Z 549.53,A -85,B 0,C 180,E1 4019.563,E2 4019.563} C_VEL
LIN {X 0,Y 536.123,Z 549.53,A -85,B 0,C 180,E1 4025.025,E2 4025.025} C_VEL
LIN {X 0,Y 536.253,Z 549.53,A -85,B 0,C 180,E1 4030.263,E2 4030.263} C_VEL
LIN {X 0,Y 536.37,Z 549.53,A -85,B 0,C 180,E1 4035.332,E2 4035.332} C_VEL
LIN {X 0,Y 536.455,Z 549.53,A -85,B 0,C 180,E1 4041.914,E2 4041.914} C_VEL
LIN {X 0,Y 536.594,Z 549.744,A -85,B 0,C 180,E1 4047.379,E2 4047.379} C_VEL
LIN {X 0,Y 544.373,Z 573.638,A -85,B 0,C 180,E1 4048.301,E2 4048.301} C_VEL
LIN {X 0,Y 543.218,Z 610.935,A -85,B 0,C 180,E1 4049.554,E2 4049.554} C_VEL
LIN {X 0,Y 541.827,Z 645.808,A -85,B 0,C 180,E1 4051.395,E2 4051.395} C_VEL
LIN {X 0,Y 540.264,Z 679.224,A -85,B 0,C 180,E1 4053.903,E2 4053.903} C_VEL
LIN {X 0,Y 538.918,Z 708.091,A -85,B 0,C 180,E1 4056.874,E2 4056.874} C_VEL
LIN {X 0,Y 537.89,Z 732.903,A -85,B 0,C 180,E1 4060.304,E2 4060.304} C_VEL
LIN {X 0,Y 537.248,Z 751.117,A -85,B 0,C 180,E1 4063.73,E2 4063.73} C_VEL
LIN {X 0,Y 536.881,Z 765.344,A -85,B 0,C 180,E1 4067.578,E2 4067.578} C_VEL
LIN {X 0,Y 536.656,Z 773.973,A -85,B 0,C 180,E1 4071.44,E2 4071.44} C_VEL
LIN {X 0,Y 536.469,Z 777.298,A -85,B 0,C 180,E1 4074.955,E2 4074.955} C_VEL
LIN {X 0,Y 536.557,Z 776.33,A -85,B 0,C 180,E1 4078.561,E2 4078.561} C_VEL
LIN {X 0,Y 536.741,Z 770.01,A -85,B 0,C 180,E1 4082.542,E2 4082.542} C_VEL
LIN {X 0,Y 536.954,Z 759.279,A -85,B 0,C 180,E1 4086.167,E2 4086.167} C_VEL
LIN {X 0,Y 537.363,Z 743.754,A -85,B 0,C 180,E1 4089.691,E2 4089.691} C_VEL
LIN {X 0,Y 538.164,Z 722.141,A -85,B 0,C 180,E1 4093.228,E2 4093.228} C_VEL
LIN {X 0,Y 539.453,Z 694.862,A -85,B 0,C 180,E1 4096.511,E2 4096.511} C_VEL
LIN {X 0,Y 541.013,Z 664.203,A -85,B 0,C 180,E1 4099.233,E2 4099.233} C_VEL
LIN {X 0,Y 542.539,Z 631.199,A -85,B 0,C 180,E1 4101.37,E2 4101.37} C_VEL
LIN {X 0,Y 543.858,Z 595.059,A -85,B 0,C 180,E1 4102.971,E2 4102.971} C_VEL
LIN {X 0,Y 543.867,Z 569.483,A -85,B 0,C 180,E1 4103.733,E2 4103.733} C_VEL
LIN {X 0,Y 536.232,Z 549.53,A -85,B 0,C 180,E1 4104.584,E2 4104.584} C_VEL
LIN {X 0,Y 536.043,Z 549.53,A -85,B 0,C 180,E1 4110.769,E2 4110.769} C_VEL
LIN {X 0,Y 536.162,Z 549.53,A -85,B 0,C 180,E1 4116.815,E2 4116.815} C_VEL
LIN {X 0,Y 536.413,Z 549.53,A -85,B 0,C 180,E1 4121.993,E2 4121.993} C_VEL
LIN {X 0,Y 536.312,Z 549.53,A -85,B 0,C 180,E1 4128.657,E2 4128.657} C_VEL
LIN {X 0,Y 536.595,Z 549.53,A -85,B 0,C 180,E1 4133.556,E2 4133.556} C_VEL
LIN {X 0,Y 536.73,Z 549.53,A -85,B 0,C 180,E1 4138.403,E2 4138.403} C_VEL
LIN {X 0,Y 536.51,Z 549.53,A -85,B 0,C 180,E1 4144.853,E2 4144.853} C_VEL
LIN {X 0,Y 536.421,Z 549.53,A -85,B 0,C 180,E1 4150.079,E2 4150.079} C_VEL
LIN {X 0,Y 536.412,Z 549.53,A -85,B 0,C 180,E1 4154.676,E2 4154.676} C_VEL
LIN {X 0,Y 536.315,Z 549.53,A -85,B 0,C 180,E1 4159.743,E2 4159.743} C_VEL
LIN {X 0,Y 536.094,Z 549.53,A -85,B 0,C 180,E1 4165.747,E2 4165.747} C_VEL
LIN {X 0,Y 536.112,Z 549.53,A -85,B 0,C 180,E1 4166.845,E2 4166.845} C_VEL
LIN {X 0,Y 532.059,Z 549.53,A -85,B 0,C 180,E1 4168.676,E2 4168.676} C_VEL
LIN {X 0,Y 528.18,Z 549.53,A -85,B 0,C 180,E1 4170.533,E2 4170.533} C_VEL
LIN {X 0,Y 528.333,Z 549.53,A -85,B 0,C 180,E1 4174.844,E2 4174.844} C_VEL
LIN {X 0,Y 528.052,Z 549.53,A -85,B 0,C 180,E1 4181.098,E2 4181.098} C_VEL
LIN {X 0,Y 528.036,Z 549.53,A -85,B 0,C 180,E1 4186.698,E2 4186.698} C_VEL
LIN {X 0,Y 528.269,Z 549.53,A -85,B 0,C 180,E1 4193.141,E2 4193.141} C_VEL
LIN {X 0,Y 528.36,Z 549.53,A -85,B 0,C 180,E1 4195.373,E2 4195.373} C_VEL
LIN {X 0,Y 540.614,Z 576.525,A -85,B 0,C 180,E1 4196.699,E2 4196.699} C_VEL
LIN {X 0,Y 540.103,Z 626.234,A -85,B 0,C 180,E1 4197.626,E2 4197.626} C_VEL
LIN {X 0,Y 538.69,Z 663.734,A -85,B 0,C 180,E1 4198.917,E2 4198.917} C_VEL
LIN {X 0,Y 536.758,Z 700.614,A -85,B 0,C 180,E1 4200.838,E2 4200.838} C_VEL
LIN {X 0,Y 534.551,Z 735.669,A -85,B 0,C 180,E1 4203.377,E2 4203.377} C_VEL
LIN {X 0,Y 532.609,Z 767.047,A -85,B 0,C 180,E1 4206.411,E2 4206.411} C_VEL
LIN {X 0,Y 530.952,Z 794.192,A -85,B 0,C 180,E1 4209.834,E2 4209.834} C_VEL
LIN {X 0,Y 529.764,Z 817.273,A -85,B 0,C 180,E1 4213.664,E2 4213.664} C_VEL
LIN {X 0,Y 529.139,Z 834.987,A -85,B 0,C 180,E1 4217.651,E2 4217.651} C_VEL
LIN {X 0,Y 528.926,Z 846.72,A -85,B 0,C 180,E1 4221.387,E2 4221.387} C_VEL
LIN {X 0,Y 528.772,Z 853.959,A -85,B 0,C 180,E1 4225.09,E2 4225.09} C_VEL
LIN {X 0,Y 528.767,Z 857.088,A -85,B 0,C 180,E1 4228.366,E2 4228.366} C_VEL
LIN {X 0,Y 528.758,Z 856.404,A -85,B 0,C 180,E1 4232.737,E2 4232.737} C_VEL
LIN {X 0,Y 528.866,Z 851.221,A -85,B 0,C 180,E1 4236.555,E2 4236.555} C_VEL
LIN {X 0,Y 528.958,Z 841.414,A -85,B 0,C 180,E1 4240.475,E2 4240.475} C_VEL
LIN {X 0,Y 529.504,Z 826.171,A -85,B 0,C 180,E1 4244.498,E2 4244.498} C_VEL
LIN {X 0,Y 530.414,Z 805.334,A -85,B 0,C 180,E1 4248.453,E2 4248.453} C_VEL
LIN {X 0,Y 531.819,Z 779.641,A -85,B 0,C 180,E1 4252.112,E2 4252.112} C_VEL
LIN {X 0,Y 533.622,Z 750.595,A -85,B 0,C 180,E1 4255.281,E2 4255.281} C_VEL
LIN {X 0,Y 535.679,Z 717.443,A -85,B 0,C 180,E1 4258.038,E2 4258.038} C_VEL
LIN {X 0,Y 537.767,Z 681.279,A -85,B 0,C 180,E1 4260.253,E2 4260.253} C_VEL
LIN {X 0,Y 539.436,Z 644.91,A -85,B 0,C 180,E1 4261.807,E2 4261.807} C_VEL
LIN {X 0,Y 540.621,Z 607.977,A -85,B 0,C 180,E1 4262.782,E2 4262.782} C_VEL
LIN {X 0,Y 540.128,Z 575.793,A -85,B 0,C 180,E1 4263.347,E2 4263.347} C_VEL
LIN {X 0,Y 528.157,Z 549.53,A -85,B 0,C 180,E1 4264.718,E2 4264.718} C_VEL
LIN {X 0,Y 528.121,Z 549.53,A -85,B 0,C 180,E1 4269.508,E2 4269.508} C_VEL
LIN {X 0,Y 528.119,Z 549.53,A -85,B 0,C 180,E1 4275.59,E2 4275.59} C_VEL
LIN {X 0,Y 528.145,Z 549.53,A -85,B 0,C 180,E1 4281.048,E2 4281.048} C_VEL
LIN {X 0,Y 528.079,Z 549.53,A -85,B 0,C 180,E1 4287.109,E2 4287.109} C_VEL
LIN {X 0,Y 528.132,Z 549.53,A -85,B 0,C 180,E1 4292.787,E2 4292.787} C_VEL
LIN {X 0,Y 528.298,Z 549.53,A -85,B 0,C 180,E1 4298.193,E2 4298.193} C_VEL
LIN {X 0,Y 528.431,Z 549.53,A -85,B 0,C 180,E1 4303.397,E2 4303.397} C_VEL
LIN {X 0,Y 528.453,Z 549.53,A -85,B 0,C 180,E1 4310.123,E2 4310.123} C_VEL
LIN {X 0,Y 528.606,Z 549.53,A -85,B 0,C 180,E1 4315.075,E2 4315.075} C_VEL
LIN {X 0,Y 528.653,Z 549.53,A -85,B 0,C 180,E1 4319.986,E2 4319.986} C_VEL
LIN {X 0,Y 528.612,Z 549.53,A -85,B 0,C 180,E1 4324.898,E2 4324.898} C_VEL
LIN {X 0,Y 528.527,Z 549.53,A -85,B 0,C 180,E1 4329.848,E2 4329.848} C_VEL
LIN {X 0,Y 528.479,Z 549.53,A -85,B 0,C 180,E1 4334.874,E2 4334.874} C_VEL
LIN {X 0,Y 528.372,Z 549.53,A -85,B 0,C 180,E1 4340.023,E2 4340.023} C_VEL
LIN {X 0,Y 528.201,Z 549.53,A -85,B 0,C 180,E1 4345.353,E2 4345.353} C_VEL
LIN {X 0,Y 528.234,Z 549.53,A -85,B 0,C 180,E1 4351.015,E2 4351.015} C_VEL
LIN {X 0,Y 528.269,Z 549.53,A -85,B 0,C 180,E1 4356.884,E2 4356.884} C_VEL
LIN {X 0,Y 528.039,Z 549.53,A -85,B 0,C 180,E1 4363.272,E2 4363.272} C_VEL
LIN {X 0,Y 528.11,Z 549.53,A -85,B 0,C 180,E1 4368.912,E2 4368.912} C_VEL
LIN {X 0,Y 528.348,Z 549.53,A -85,B 0,C 180,E1 4375.163,E2 4375.163} C_VEL
LIN {X 0,Y 528.238,Z 549.53,A -85,B 0,C 180,E1 4380.944,E2 4380.944} C_VEL
LIN {X 0,Y 528.23,Z 549.53,A -85,B 0,C 180,E1 4386.424,E2 4386.424} C_VEL
LIN {X 0,Y 528.379,Z 549.53,A -85,B 0,C 180,E1 4391.689,E2 4391.689} C_VEL
LIN {X 0,Y 528.475,Z 549.53,A -85,B 0,C 180,E1 4396.794,E2 4396.794} C_VEL
LIN {X 0,Y 528.565,Z 549.53,A -85,B 0,C 180,E1 4401.792,E2 4401.792} C_VEL
LIN {X 0,Y 528.741,Z 549.53,A -85,B 0,C 180,E1 4406.879,E2 4406.879} C_VEL
LIN {X 0,Y 537.316,Z 576.062,A -85,B 0,C 180,E1 4407.976,E2 4407.976} C_VEL
LIN {X 0,Y 536.008,Z 613.143,A -85,B 0,C 180,E1 4409.273,E2 4409.273} C_VEL
LIN {X 0,Y 534.417,Z 648.55,A -85,B 0,C 180,E1 4411.212,E2 4411.212} C_VEL
LIN {X 0,Y 532.686,Z 681.14,A -85,B 0,C 180,E1 4413.755,E2 4413.755} C_VEL
LIN {X 0,Y 531.219,Z 709.24,A -85,B 0,C 180,E1 4416.728,E2 4416.728} C_VEL
LIN {X 0,Y 530.121,Z 733.133,A -85,B 0,C 180,E1 4420.106,E2 4420.106} C_VEL
LIN {X 0,Y 529.369,Z 751.957,A -85,B 0,C 180,E1 4423.742,E2 4423.742} C_VEL
LIN {X 0,Y 528.999,Z 765.507,A -85,B 0,C 180,E1 4427.511,E2 4427.511} C_VEL
LIN {X 0,Y 528.831,Z 773.256,A -85,B 0,C 180,E1 4430.895,E2 4430.895} C_VEL
LIN {X 0,Y 528.55,Z 776.851,A -85,B 0,C 180,E1 4434.056,E2 4434.056} C_VEL
LIN {X 0,Y 528.601,Z 776.88,A -85,B 0,C 180,E1 4437.808,E2 4437.808} C_VEL
LIN {X 0,Y 528.82,Z 772.965,A -85,B 0,C 180,E1 4441.171,E2 4441.171} C_VEL
LIN {X 0,Y 529.065,Z 763.395,A -85,B 0,C 180,E1 4445.098,E2 4445.098} C_VEL
LIN {X 0,Y 529.419,Z 748.938,A -85,B 0,C 180,E1 4448.833,E2 4448.833} C_VEL
LIN {X 0,Y 530.208,Z 729.201,A -85,B 0,C 180,E1 4452.432,E2 4452.432} C_VEL
LIN {X 0,Y 531.543,Z 702.925,A -85,B 0,C 180,E1 4455.931,E2 4455.931} C_VEL
LIN {X 0,Y 533.08,Z 673.829,A -85,B 0,C 180,E1 4458.797,E2 4458.797} C_VEL
LIN {X 0,Y 534.854,Z 641.233,A -85,B 0,C 180,E1 4461.157,E2 4461.157} C_VEL
LIN {X 0,Y 536.437,Z 605.223,A -85,B 0,C 180,E1 4462.97,E2 4462.97} C_VEL
LIN {X 0,Y 536.738,Z 571.558,A -85,B 0,C 180,E1 4464.086,E2 4464.086} C_VEL
LIN {X 0,Y 528.223,Z 549.53,A -85,B 0,C 180,E1 4465.113,E2 4465.113} C_VEL
LIN {X 0,Y 528.161,Z 549.53,A -85,B 0,C 180,E1 4470.964,E2 4470.964} C_VEL
LIN {X 0,Y 528.208,Z 549.53,A -85,B 0,C 180,E1 4476.445,E2 4476.445} C_VEL
LIN {X 0,Y 528.475,Z 549.53,A -85,B 0,C 180,E1 4481.713,E2 4481.713} C_VEL
LIN {X 0,Y 528.369,Z 549.53,A -85,B 0,C 180,E1 4488.484,E2 4488.484} C_VEL
LIN {X 0,Y 528.671,Z 549.53,A -85,B 0,C 180,E1 4493.459,E2 4493.459} C_VEL
LIN {X 0,Y 528.82,Z 549.53,A -85,B 0,C 180,E1 4498.379,E2 4498.379} C_VEL
LIN {X 0,Y 528.612,Z 549.53,A -85,B 0,C 180,E1 4504.925,E2 4504.925} C_VEL
LIN {X 0,Y 528.54,Z 549.53,A -85,B 0,C 180,E1 4509.875,E2 4509.875} C_VEL
LIN {X 0,Y 528.494,Z 549.53,A -85,B 0,C 180,E1 4514.901,E2 4514.901} C_VEL
LIN {X 0,Y 528.384,Z 549.53,A -85,B 0,C 180,E1 4520.052,E2 4520.052} C_VEL
LIN {X 0,Y 528.217,Z 549.53,A -85,B 0,C 180,E1 4525.382,E2 4525.382} C_VEL
LIN {X 0,Y 528.18,Z 549.53,A -85,B 0,C 180,E1 4530.533,E2 4530.533} C_VEL
LIN {X 0,Y 525.735,Z 549.53,A -85,B 0,C 180,E1 4531.937,E2 4531.937} C_VEL
LIN {X 0,Y 520.303,Z 549.53,A -85,B 0,C 180,E1 4534.283,E2 4534.283} C_VEL
LIN {X 0,Y 520.209,Z 549.53,A -85,B 0,C 180,E1 4539.662,E2 4539.662} C_VEL
LIN {X 0,Y 520.106,Z 549.53,A -85,B 0,C 180,E1 4545.869,E2 4545.869} C_VEL
LIN {X 0,Y 520.245,Z 549.53,A -85,B 0,C 180,E1 4551.556,E2 4551.556} C_VEL
LIN {X 0,Y 520.409,Z 549.812,A -85,B 0,C 180,E1 4554.784,E2 4554.784} C_VEL
LIN {X 0,Y 534.081,Z 579.518,A -85,B 0,C 180,E1 4556.284,E2 4556.284} C_VEL
LIN {X 0,Y 533.396,Z 625.826,A -85,B 0,C 180,E1 4557.156,E2 4557.156} C_VEL
LIN {X 0,Y 531.816,Z 664.481,A -85,B 0,C 180,E1 4558.507,E2 4558.507} C_VEL
LIN {X 0,Y 529.669,Z 701.743,A -85,B 0,C 180,E1 4560.488,E2 4560.488} C_VEL
LIN {X 0,Y 527.218,Z 736.924,A -85,B 0,C 180,E1 4563.092,E2 4563.092} C_VEL
LIN {X 0,Y 525.01,Z 768.959,A -85,B 0,C 180,E1 4566.273,E2 4566.273} C_VEL
LIN {X 0,Y 523.231,Z 795.714,A -85,B 0,C 180,E1 4569.753,E2 4569.753} C_VEL
LIN {X 0,Y 521.941,Z 818.358,A -85,B 0,C 180,E1 4573.628,E2 4573.628} C_VEL
LIN {X 0,Y 521.295,Z 834.988,A -85,B 0,C 180,E1 4577.462,E2 4577.462} C_VEL
LIN {X 0,Y 521.057,Z 846.72,A -85,B 0,C 180,E1 4581.256,E2 4581.256} C_VEL
LIN {X 0,Y 520.876,Z 853.959,A -85,B 0,C 180,E1 4585.015,E2 4585.015} C_VEL
LIN {X 0,Y 520.881,Z 857.088,A -85,B 0,C 180,E1 4588.341,E2 4588.341} C_VEL
LIN {X 0,Y 521,Z 857.087,A -85,B 0,C 180,E1 4591.661,E2 4591.661} C_VEL
LIN {X 0,Y 520.999,Z 852.753,A -85,B 0,C 180,E1 4595.82,E2 4595.82} C_VEL
LIN {X 0,Y 521.101,Z 843.121,A -85,B 0,C 180,E1 4600.073,E2 4600.073} C_VEL
LIN {X 0,Y 521.653,Z 827.176,A -85,B 0,C 180,E1 4604.5,E2 4604.5} C_VEL
LIN {X 0,Y 522.646,Z 806.654,A -85,B 0,C 180,E1 4608.519,E2 4608.519} C_VEL
LIN {X 0,Y 524.251,Z 780.279,A -85,B 0,C 180,E1 4612.367,E2 4612.367} C_VEL
LIN {X 0,Y 526.326,Z 750.155,A -85,B 0,C 180,E1 4615.7,E2 4615.7} C_VEL
LIN {X 0,Y 528.589,Z 716.779,A -85,B 0,C 180,E1 4618.498,E2 4618.498} C_VEL
LIN {X 0,Y 530.863,Z 680.844,A -85,B 0,C 180,E1 4620.713,E2 4620.713} C_VEL
LIN {X 0,Y 532.713,Z 643.8,A -85,B 0,C 180,E1 4622.297,E2 4622.297} C_VEL
LIN {X 0,Y 534.082,Z 606.039,A -85,B 0,C 180,E1 4623.271,E2 4623.271} C_VEL
LIN {X 0,Y 533.494,Z 578.419,A -85,B 0,C 180,E1 4623.775,E2 4623.775} C_VEL
LIN {X 0,Y 520.204,Z 549.53,A -85,B 0,C 180,E1 4625.286,E2 4625.286} C_VEL
LIN {X 0,Y 520.16,Z 549.53,A -85,B 0,C 180,E1 4631.033,E2 4631.033} C_VEL
LIN {X 0,Y 520.198,Z 549.53,A -85,B 0,C 180,E1 4636.488,E2 4636.488} C_VEL
LIN {X 0,Y 520.203,Z 549.53,A -85,B 0,C 180,E1 4642.463,E2 4642.463} C_VEL
LIN {X 0,Y 520.18,Z 549.53,A -85,B 0,C 180,E1 4648.514,E2 4648.514} C_VEL
LIN {X 0,Y 520.246,Z 549.53,A -85,B 0,C 180,E1 4654.2,E2 4654.2} C_VEL
LIN {X 0,Y 520.447,Z 549.53,A -85,B 0,C 180,E1 4659.629,E2 4659.629} C_VEL
LIN {X 0,Y 520.356,Z 549.53,A -85,B 0,C 180,E1 4664.86,E2 4664.86} C_VEL
LIN {X 0,Y 520.553,Z 549.53,A -85,B 0,C 180,E1 4670.277,E2 4670.277} C_VEL
LIN {X 0,Y 520.7,Z 549.53,A -85,B 0,C 180,E1 4675,E2 4675} C_VEL
LIN {X 0,Y 520.765,Z 549.53,A -85,B 0,C 180,E1 4679.986,E2 4679.986} C_VEL
LIN {X 0,Y 520.698,Z 549.53,A -85,B 0,C 180,E1 4684.973,E2 4684.973} C_VEL
LIN {X 0,Y 520.62,Z 549.53,A -85,B 0,C 180,E1 4689.999,E2 4689.999} C_VEL
LIN {X 0,Y 520.545,Z 549.53,A -85,B 0,C 180,E1 4695.106,E2 4695.106} C_VEL
